LIN {X 0,Y 373.956,Z 1100.228,A -85,B 0,C 180,E1 19319.905,E2 19319.905} C_VEL
LIN {X 0,Y 365.783,Z 1123.311,A -85,B 0,C 180,E1 19326.825,E2 19326.825} C_VEL
LIN {X 0,Y 361.232,Z 1139.651,A -85,B 0,C 180,E1 19333.998,E2 19333.998} C_VEL
LIN {X 0,Y 359.65,Z 1148.795,A -85,B 0,C 180,E1 19340.296,E2 19340.296} C_VEL
LIN {X 0,Y 359.245,Z 1152.82,A -85,B 0,C 180,E1 19345.159,E2 19345.159} C_VEL
LIN {X 0,Y 359.425,Z 1154.198,A -85,B 0,C 180,E1 19349.998,E2 19349.998} C_VEL
LIN {X 0,Y 359.256,Z 1152.829,A -85,B 0,C 180,E1 19354.837,E2 19354.837} C_VEL
LIN {X 0,Y 359.821,Z 1147.421,A -85,B 0,C 180,E1 19360.921,E2 19360.921} C_VEL
LIN {X 0,Y 362.025,Z 1136.467,A -85,B 0,C 180,E1 19367.662,E2 19367.662} C_VEL
LIN {X 0,Y 366.908,Z 1119.796,A -85,B 0,C 180,E1 19374.388,E2 19374.388} C_VEL
LIN {X 0,Y 374.76,Z 1097.852,A -85,B 0,C 180,E1 19380.69,E2 19380.69} C_VEL
LIN {X 0,Y 385.507,Z 1070.168,A -85,B 0,C 180,E1 19386.483,E2 19386.483} C_VEL
LIN {X 0,Y 398.345,Z 1037.029,A -85,B 0,C 180,E1 19391.528,E2 19391.528} C_VEL
LIN {X 0,Y 411.863,Z 998.645,A -85,B 0,C 180,E1 19395.754,E2 19395.754} C_VEL
LIN {X 0,Y 424.268,Z 957.523,A -85,B 0,C 180,E1 19398.972,E2 19398.972} C_VEL
LIN {X 0,Y 433.607,Z 917.598,A -85,B 0,C 180,E1 19401.2,E2 19401.2} C_VEL
LIN {X 0,Y 431.056,Z 908.486,A -85,B 0,C 180,E1 19402.307,E2 19402.307} C_VEL
LIN {X 0,Y 426.576,Z 900.935,A -85,B 0,C 180,E1 19403.608,E2 19403.608} C_VEL
LIN {X 0,Y 417.797,Z 890.205,A -85,B 0,C 180,E1 19405.959,E2 19405.959} C_VEL
LIN {X 0,Y 405.491,Z 863.569,A -85,B 0,C 180,E1 19410.288,E2 19410.288} C_VEL
LIN {X 0,Y 391.387,Z 839.153,A -85,B 0,C 180,E1 19415.267,E2 19415.267} C_VEL
LIN {X 0,Y 377.889,Z 819.617,A -85,B 0,C 180,E1 19420.846,E2 19420.846} C_VEL
LIN {X 0,Y 371.927,Z 812.012,A -85,B 0,C 180,E1 19423.898,E2 19423.898} C_VEL
LIN {X 0,Y 367.631,Z 805.669,A -85,B 0,C 180,E1 19426.606,E2 19426.606} C_VEL
LIN {X 0,Y 363.551,Z 800.282,A -85,B 0,C 180,E1 19429.732,E2 19429.732} C_VEL
LIN {X 0,Y 362.215,Z 798.402,A -85,B 0,C 180,E1 19430.985,E2 19430.985} C_VEL
LIN {X 0,Y 357.922,Z 792.601,A -85,B 0,C 180,E1 19436.9,E2 19436.9} C_VEL
LIN {X 0,Y 357.785,Z 791.099,A -85,B 0,C 180,E1 19437.582,E2 19437.582} C_VEL
LIN {X 0,Y 357.664,Z 791.872,A -85,B 0,C 180,E1 19445.486,E2 19445.486} C_VEL
LIN {X 0,Y 360.859,Z 797.744,A -85,B 0,C 180,E1 19450.899,E2 19450.899} C_VEL
LIN {X 0,Y 363.277,Z 799.765,A -85,B 0,C 180,E1 19453.203,E2 19453.203} C_VEL
LIN {X 0,Y 366.794,Z 805.247,A -85,B 0,C 180,E1 19456.044,E2 19456.044} C_VEL
LIN {X 0,Y 368.948,Z 807.739,A -85,B 0,C 180,E1 19457.467,E2 19457.467} C_VEL
LIN {X 0,Y 374.683,Z 815.764,A -85,B 0,C 180,E1 19460.76,E2 19460.76} C_VEL
LIN {X 0,Y 383.493,Z 827.748,A -85,B 0,C 180,E1 19464.796,E2 19464.796} C_VEL
LIN {X 0,Y 398.322,Z 850.048,A -85,B 0,C 180,E1 19470.272,E2 19470.272} C_VEL
LIN {X 0,Y 412.31,Z 876.094,A -85,B 0,C 180,E1 19475.03,E2 19475.03} C_VEL
LIN {X 0,Y 424.367,Z 905.945,A -85,B 0,C 180,E1 19479.392,E2 19479.392} C_VEL
LIN {X 0,Y 428.186,Z 921.116,A -85,B 0,C 180,E1 19481.238,E2 19481.238} C_VEL
LIN {X 0,Y 417.887,Z 960.689,A -85,B 0,C 180,E1 19483.521,E2 19483.521} C_VEL
LIN {X 0,Y 406.177,Z 996.477,A -85,B 0,C 180,E1 19486.442,E2 19486.442} C_VEL
LIN {X 0,Y 392.908,Z 1031.099,A -85,B 0,C 180,E1 19490.39,E2 19490.39} C_VEL
LIN {X 0,Y 380.116,Z 1061.22,A -85,B 0,C 180,E1 19495.164,E2 19495.164} C_VEL
LIN {X 0,Y 368.183,Z 1087.867,A -85,B 0,C 180,E1 19501.085,E2 19501.085} C_VEL
LIN {X 0,Y 359.507,Z 1108.593,A -85,B 0,C 180,E1 19507.711,E2 19507.711} C_VEL
LIN {X 0,Y 354.448,Z 1122.693,A -85,B 0,C 180,E1 19514.392,E2 19514.392} C_VEL
LIN {X 0,Y 352.341,Z 1130.443,A -85,B 0,C 180,E1 19520.097,E2 19520.097} C_VEL
LIN {X 0,Y 351.551,Z 1134.292,A -85,B 0,C 180,E1 19525.057,E2 19525.057} C_VEL
LIN {X 0,Y 351.584,Z 1135.551,A -85,B 0,C 180,E1 19530.002,E2 19530.002} C_VEL
LIN {X 0,Y 351.61,Z 1134.245,A -85,B 0,C 180,E1 19534.946,E2 19534.946} C_VEL
LIN {X 0,Y 352.649,Z 1128.889,A -85,B 0,C 180,E1 19541.15,E2 19541.15} C_VEL
LIN {X 0,Y 355.894,Z 1118.129,A -85,B 0,C 180,E1 19547.981,E2 19547.981} C_VEL
LIN {X 0,Y 362.33,Z 1101.558,A -85,B 0,C 180,E1 19554.721,E2 19554.721} C_VEL
LIN {X 0,Y 372.526,Z 1078.136,A -85,B 0,C 180,E1 19561.211,E2 19561.211} C_VEL
LIN {X 0,Y 384.637,Z 1050.732,A -85,B 0,C 180,E1 19566.572,E2 19566.572} C_VEL
LIN {X 0,Y 398.251,Z 1017.644,A -85,B 0,C 180,E1 19571.2,E2 19571.2} C_VEL
LIN {X 0,Y 411.718,Z 980.096,A -85,B 0,C 180,E1 19574.923,E2 19574.923} C_VEL
LIN {X 0,Y 423.676,Z 939.446,A -85,B 0,C 180,E1 19577.719,E2 19577.719} C_VEL
LIN {X 0,Y 428.181,Z 918.706,A -85,B 0,C 180,E1 19578.835,E2 19578.835} C_VEL
LIN {X 0,Y 417.88,Z 888.908,A -85,B 0,C 180,E1 19582.883,E2 19582.883} C_VEL
LIN {X 0,Y 404.192,Z 860.481,A -85,B 0,C 180,E1 19587.547,E2 19587.547} C_VEL
LIN {X 0,Y 389.923,Z 837.253,A -85,B 0,C 180,E1 19592.513,E2 19592.513} C_VEL
LIN {X 0,Y 377.483,Z 819.326,A -85,B 0,C 180,E1 19597.664,E2 19597.664} C_VEL
LIN {X 0,Y 372.107,Z 812.286,A -85,B 0,C 180,E1 19600.401,E2 19600.401} C_VEL
LIN {X 0,Y 367.521,Z 805.745,A -85,B 0,C 180,E1 19603.219,E2 19603.219} C_VEL
LIN {X 0,Y 363.319,Z 800.256,A -85,B 0,C 180,E1 19606.402,E2 19606.402} C_VEL
LIN {X 0,Y 362.197,Z 798.481,A -85,B 0,C 180,E1 19607.448,E2 19607.448} C_VEL
LIN {X 0,Y 357.808,Z 792.997,A -85,B 0,C 180,E1 19613.093,E2 19613.093} C_VEL
LIN {X 0,Y 357.566,Z 791.207,A -85,B 0,C 180,E1 19613.969,E2 19613.969} C_VEL
LIN {X 0,Y 357.77,Z 791.665,A -85,B 0,C 180,E1 19623.253,E2 19623.253} C_VEL
LIN {X 0,Y 360.689,Z 797.51,A -85,B 0,C 180,E1 19627.837,E2 19627.837} C_VEL
LIN {X 0,Y 363.41,Z 799.856,A -85,B 0,C 180,E1 19630.348,E2 19630.348} C_VEL
LIN {X 0,Y 367.37,Z 805.514,A -85,B 0,C 180,E1 19633.404,E2 19633.404} C_VEL
LIN {X 0,Y 369.332,Z 808.368,A -85,B 0,C 180,E1 19634.694,E2 19634.694} C_VEL
LIN {X 0,Y 374.696,Z 815.689,A -85,B 0,C 180,E1 19637.72,E2 19637.72} C_VEL
LIN {X 0,Y 383.778,Z 828.216,A -85,B 0,C 180,E1 19641.864,E2 19641.864} C_VEL
LIN {X 0,Y 397.292,Z 848.846,A -85,B 0,C 180,E1 19646.917,E2 19646.917} C_VEL
LIN {X 0,Y 411.35,Z 875.442,A -85,B 0,C 180,E1 19651.804,E2 19651.804} C_VEL
LIN {X 0,Y 423.261,Z 905.411,A -85,B 0,C 180,E1 19656.19,E2 19656.19} C_VEL
LIN {X 0,Y 427.768,Z 921.449,A -85,B 0,C 180,E1 19658.22,E2 19658.22} C_VEL
LIN {X 0,Y 417.52,Z 961.645,A -85,B 0,C 180,E1 19660.513,E2 19660.513} C_VEL
LIN {X 0,Y 405.27,Z 1000.897,A -85,B 0,C 180,E1 19663.695,E2 19663.695} C_VEL
LIN {X 0,Y 391.626,Z 1038.299,A -85,B 0,C 180,E1 19667.909,E2 19667.909} C_VEL
LIN {X 0,Y 378.356,Z 1071.449,A -85,B 0,C 180,E1 19673.078,E2 19673.078} C_VEL
LIN {X 0,Y 366.86,Z 1099.983,A -85,B 0,C 180,E1 19679.261,E2 19679.261} C_VEL
LIN {X 0,Y 358.287,Z 1123.082,A -85,B 0,C 180,E1 19686.31,E2 19686.31} C_VEL
LIN {X 0,Y 353.392,Z 1139.77,A -85,B 0,C 180,E1 19693.816,E2 19693.816} C_VEL
LIN {X 0,Y 351.787,Z 1148.584,A -85,B 0,C 180,E1 19700.077,E2 19700.077} C_VEL
LIN {X 0,Y 351.344,Z 1152.612,A -85,B 0,C 180,E1 19705.05,E2 19705.05} C_VEL
LIN {X 0,Y 351.526,Z 1153.991,A -85,B 0,C 180,E1 19709.998,E2 19709.998} C_VEL
LIN {X 0,Y 351.354,Z 1152.621,A -85,B 0,C 180,E1 19714.946,E2 19714.946} C_VEL
LIN {X 0,Y 351.953,Z 1147.208,A -85,B 0,C 180,E1 19721.168,E2 19721.168} C_VEL
LIN {X 0,Y 354.33,Z 1136.25,A -85,B 0,C 180,E1 19728.058,E2 19728.058} C_VEL
LIN {X 0,Y 359.478,Z 1119.569,A -85,B 0,C 180,E1 19734.926,E2 19734.926} C_VEL
LIN {X 0,Y 367.707,Z 1097.609,A -85,B 0,C 180,E1 19741.345,E2 19741.345} C_VEL
LIN {X 0,Y 378.945,Z 1069.961,A -85,B 0,C 180,E1 19747.209,E2 19747.209} C_VEL
LIN {X 0,Y 392.299,Z 1036.729,A -85,B 0,C 180,E1 19752.316,E2 19752.316} C_VEL
LIN {X 0,Y 406.23,Z 998.283,A -85,B 0,C 180,E1 19756.577,E2 19756.577} C_VEL
LIN {X 0,Y 419.021,Z 957.147,A -85,B 0,C 180,E1 19759.799,E2 19759.799} C_VEL
LIN {X 0,Y 427.819,Z 920.28,A -85,B 0,C 180,E1 19761.9,E2 19761.9} C_VEL
LIN {X 0,Y 417.931,Z 890.491,A -85,B 0,C 180,E1 19765.913,E2 19765.913} C_VEL
LIN {X 0,Y 417.797,Z 890.205,A -85,B 0,C 180,E1 19765.959,E2 19765.959} C_VEL
LIN {X 0,Y 414.753,Z 885.487,A -85,B 0,C 180,E1 19766.885,E2 19766.885} C_VEL
LIN {X 0,Y 404.818,Z 875.598,A -85,B 0,C 180,E1 19769.67,E2 19769.67} C_VEL
LIN {X 0,Y 404.141,Z 874.327,A -85,B 0,C 180,E1 19769.908,E2 19769.908} C_VEL
LIN {X 0,Y 390.792,Z 849.549,A -85,B 0,C 180,E1 19774.923,E2 19774.923} C_VEL
LIN {X 0,Y 379.056,Z 831.63,A -85,B 0,C 180,E1 19779.768,E2 19779.768} C_VEL
LIN {X 0,Y 370.576,Z 819.735,A -85,B 0,C 180,E1 19784.066,E2 19784.066} C_VEL
LIN {X 0,Y 365.782,Z 813.016,A -85,B 0,C 180,E1 19787.146,E2 19787.146} C_VEL
LIN {X 0,Y 361.886,Z 806.955,A -85,B 0,C 180,E1 19790.369,E2 19790.369} C_VEL
LIN {X 0,Y 356.82,Z 800.076,A -85,B 0,C 180,E1 19797.271,E2 19797.271} C_VEL
LIN {X 0,Y 356.387,Z 798.849,A -85,B 0,C 180,E1 19798.791,E2 19798.791} C_VEL
LIN {X 0,Y 356.618,Z 799.725,A -85,B 0,C 180,E1 19805.296,E2 19805.296} C_VEL
LIN {X 0,Y 359.918,Z 805.614,A -85,B 0,C 180,E1 19810.928,E2 19810.928} C_VEL
LIN {X 0,Y 361.974,Z 807.59,A -85,B 0,C 180,E1 19812.943,E2 19812.943} C_VEL
LIN {X 0,Y 365.87,Z 813.166,A -85,B 0,C 180,E1 19816.086,E2 19816.086} C_VEL
LIN {X 0,Y 373.131,Z 823.471,A -85,B 0,C 180,E1 19820.507,E2 19820.507} C_VEL
LIN {X 0,Y 381.532,Z 835.16,A -85,B 0,C 180,E1 19824.45,E2 19824.45} C_VEL
LIN {X 0,Y 395.223,Z 856.602,A -85,B 0,C 180,E1 19829.82,E2 19829.82} C_VEL
LIN {X 0,Y 408.571,Z 882.567,A -85,B 0,C 180,E1 19834.645,E2 19834.645} C_VEL
LIN {X 0,Y 419.409,Z 910.851,A -85,B 0,C 180,E1 19838.886,E2 19838.886} C_VEL
LIN {X 0,Y 422.643,Z 923.525,A -85,B 0,C 180,E1 19840.525,E2 19840.525} C_VEL
LIN {X 0,Y 411.782,Z 963.336,A -85,B 0,C 180,E1 19842.877,E2 19842.877} C_VEL
LIN {X 0,Y 399.286,Z 999.96,A -85,B 0,C 180,E1 19845.975,E2 19845.975} C_VEL
LIN {X 0,Y 386.152,Z 1032.812,A -85,B 0,C 180,E1 19849.836,E2 19849.836} C_VEL
LIN {X 0,Y 373.24,Z 1062.126,A -85,B 0,C 180,E1 19854.592,E2 19854.592} C_VEL
LIN {X 0,Y 361.146,Z 1088.094,A -85,B 0,C 180,E1 19860.467,E2 19860.467} C_VEL
LIN {X 0,Y 352.084,Z 1108.811,A -85,B 0,C 180,E1 19867.215,E2 19867.215} C_VEL
LIN {X 0,Y 346.742,Z 1122.898,A -85,B 0,C 180,E1 19874.031,E2 19874.031} C_VEL
LIN {X 0,Y 344.182,Z 1131.817,A -85,B 0,C 180,E1 19881.139,E2 19881.139} C_VEL
LIN {X 0,Y 343.604,Z 1135.449,A -85,B 0,C 180,E1 19887.475,E2 19887.475} C_VEL
LIN {X 0,Y 343.67,Z 1135.428,A -85,B 0,C 180,E1 19892.529,E2 19892.529} C_VEL
LIN {X 0,Y 344.122,Z 1132.272,A -85,B 0,C 180,E1 19898.251,E2 19898.251} C_VEL
LIN {X 0,Y 346.349,Z 1123.943,A -85,B 0,C 180,E1 19905.22,E2 19905.22} C_VEL
LIN {X 0,Y 352.168,Z 1108.548,A -85,B 0,C 180,E1 19912.784,E2 19912.784} C_VEL
LIN {X 0,Y 361.342,Z 1087.725,A -85,B 0,C 180,E1 19919.52,E2 19919.52} C_VEL
LIN {X 0,Y 373.954,Z 1060.341,A -85,B 0,C 180,E1 19925.646,E2 19925.646} C_VEL
LIN {X 0,Y 388.096,Z 1028.24,A -85,B 0,C 180,E1 19930.669,E2 19930.669} C_VEL
LIN {X 0,Y 402.094,Z 992.251,A -85,B 0,C 180,E1 19934.66,E2 19934.66} C_VEL
LIN {X 0,Y 414.776,Z 953.143,A -85,B 0,C 180,E1 19937.711,E2 19937.711} C_VEL
LIN {X 0,Y 422.617,Z 922.16,A -85,B 0,C 180,E1 19939.467,E2 19939.467} C_VEL
LIN {X 0,Y 412.652,Z 892.425,A -85,B 0,C 180,E1 19943.666,E2 19943.666} C_VEL
LIN {X 0,Y 400.208,Z 865.768,A -85,B 0,C 180,E1 19948.226,E2 19948.226} C_VEL
LIN {X 0,Y 386.717,Z 843.189,A -85,B 0,C 180,E1 19953.213,E2 19953.213} C_VEL
LIN {X 0,Y 375.38,Z 826.412,A -85,B 0,C 180,E1 19958.148,E2 19958.148} C_VEL
LIN {X 0,Y 370.2,Z 819.464,A -85,B 0,C 180,E1 19960.88,E2 19960.88} C_VEL
LIN {X 0,Y 365.691,Z 813.099,A -85,B 0,C 180,E1 19963.752,E2 19963.752} C_VEL
LIN {X 0,Y 361.772,Z 807.296,A -85,B 0,C 180,E1 19966.913,E2 19966.913} C_VEL
LIN {X 0,Y 356.662,Z 800.295,A -85,B 0,C 180,E1 19973.552,E2 19973.552} C_VEL
LIN {X 0,Y 356.158,Z 798.839,A -85,B 0,C 180,E1 19975.11,E2 19975.11} C_VEL
LIN {X 0,Y 356.714,Z 799.636,A -85,B 0,C 180,E1 19983.11,E2 19983.11} C_VEL
LIN {X 0,Y 360.019,Z 805.576,A -85,B 0,C 180,E1 19988.156,E2 19988.156} C_VEL
LIN {X 0,Y 362.076,Z 807.594,A -85,B 0,C 180,E1 19990.082,E2 19990.082} C_VEL
LIN {X 0,Y 366.184,Z 813.294,A -85,B 0,C 180,E1 19993.296,E2 19993.296} C_VEL
LIN {X 0,Y 373.149,Z 823.441,A -85,B 0,C 180,E1 19997.491,E2 19997.491} C_VEL
LIN {X 0,Y 381.743,Z 835.576,A -85,B 0,C 180,E1 20001.528,E2 20001.528} C_VEL
LIN {X 0,Y 394.839,Z 856.498,A -85,B 0,C 180,E1 20006.712,E2 20006.712} C_VEL
LIN {X 0,Y 408.266,Z 883.5,A -85,B 0,C 180,E1 20011.681,E2 20011.681} C_VEL
LIN {X 0,Y 418.825,Z 911.999,A -85,B 0,C 180,E1 20015.909,E2 20015.909} C_VEL
LIN {X 0,Y 421.842,Z 925.41,A -85,B 0,C 180,E1 20017.579,E2 20017.579} C_VEL
LIN {X 0,Y 410.357,Z 967.994,A -85,B 0,C 180,E1 20020.141,E2 20020.141} C_VEL
LIN {X 0,Y 397.869,Z 1005.569,A -85,B 0,C 180,E1 20023.349,E2 20023.349} C_VEL
LIN {X 0,Y 384.76,Z 1040.072,A -85,B 0,C 180,E1 20027.384,E2 20027.384} C_VEL
LIN {X 0,Y 371.326,Z 1072.396,A -85,B 0,C 180,E1 20032.554,E2 20032.554} C_VEL
LIN {X 0,Y 359.735,Z 1099.736,A -85,B 0,C 180,E1 20038.583,E2 20038.583} C_VEL
LIN {X 0,Y 351.295,Z 1121.451,A -85,B 0,C 180,E1 20045.277,E2 20045.277} C_VEL
LIN {X 0,Y 346.242,Z 1137.175,A -85,B 0,C 180,E1 20052.16,E2 20052.16} C_VEL
LIN {X 0,Y 344.148,Z 1146.969,A -85,B 0,C 180,E1 20058.571,E2 20058.571} C_VEL
LIN {X 0,Y 343.457,Z 1152.404,A -85,B 0,C 180,E1 20064.936,E2 20064.936} C_VEL
LIN {X 0,Y 343.654,Z 1153.784,A -85,B 0,C 180,E1 20069.998,E2 20069.998} C_VEL
LIN {X 0,Y 343.464,Z 1152.414,A -85,B 0,C 180,E1 20075.059,E2 20075.059} C_VEL
LIN {X 0,Y 344.118,Z 1146.997,A -85,B 0,C 180,E1 20081.426,E2 20081.426} C_VEL
LIN {X 0,Y 346.636,Z 1136.033,A -85,B 0,C 180,E1 20088.473,E2 20088.473} C_VEL
LIN {X 0,Y 352.107,Z 1119.343,A -85,B 0,C 180,E1 20095.485,E2 20095.485} C_VEL
LIN {X 0,Y 360.712,Z 1097.368,A -85,B 0,C 180,E1 20102.024,E2 20102.024} C_VEL
LIN {X 0,Y 372.498,Z 1069.702,A -85,B 0,C 180,E1 20107.965,E2 20107.965} C_VEL
LIN {X 0,Y 386.02,Z 1037.209,A -85,B 0,C 180,E1 20113.03,E2 20113.03} C_VEL
LIN {X 0,Y 400.418,Z 998.783,A -85,B 0,C 180,E1 20117.342,E2 20117.342} C_VEL
LIN {X 0,Y 413.86,Z 956.676,A -85,B 0,C 180,E1 20120.657,E2 20120.657} C_VEL
LIN {X 0,Y 422.114,Z 923.436,A -85,B 0,C 180,E1 20122.577,E2 20122.577} C_VEL
LIN {X 0,Y 412.89,Z 894.546,A -85,B 0,C 180,E1 20126.615,E2 20126.615} C_VEL
LIN {X 0,Y 404.141,Z 874.327,A -85,B 0,C 180,E1 20129.908,E2 20129.908} C_VEL
LIN {X 0,Y 399.335,Z 868.608,A -85,B 0,C 180,E1 20131.445,E2 20131.445} C_VEL
LIN {X 0,Y 390.73,Z 861.226,A -85,B 0,C 180,E1 20134.206,E2 20134.206} C_VEL
LIN {X 0,Y 377.96,Z 840.111,A -85,B 0,C 180,E1 20139.686,E2 20139.686} C_VEL
LIN {X 0,Y 368.6,Z 826.875,A -85,B 0,C 180,E1 20144.59,E2 20144.59} C_VEL
LIN {X 0,Y 364.127,Z 820.46,A -85,B 0,C 180,E1 20147.577,E2 20147.577} C_VEL
LIN {X 0,Y 359.657,Z 813.776,A -85,B 0,C 180,E1 20151.531,E2 20151.531} C_VEL
LIN {X 0,Y 355.734,Z 807.55,A -85,B 0,C 180,E1 20157.645,E2 20157.645} C_VEL
LIN {X 0,Y 355.545,Z 807.004,A -85,B 0,C 180,E1 20164.827,E2 20164.827} C_VEL
LIN {X 0,Y 358.431,Z 813.129,A -85,B 0,C 180,E1 20170.358,E2 20170.358} C_VEL
LIN {X 0,Y 360.688,Z 815.356,A -85,B 0,C 180,E1 20172.684,E2 20172.684} C_VEL
LIN {X 0,Y 365.08,Z 821.214,A -85,B 0,C 180,E1 20176.218,E2 20176.218} C_VEL
LIN {X 0,Y 375.393,Z 836.314,A -85,B 0,C 180,E1 20182.189,E2 20182.189} C_VEL
LIN {X 0,Y 387.289,Z 855.022,A -85,B 0,C 180,E1 20187.452,E2 20187.452} C_VEL
LIN {X 0,Y 400.473,Z 879.378,A -85,B 0,C 180,E1 20192.594,E2 20192.594} C_VEL
LIN {X 0,Y 411.5,Z 906.731,A -85,B 0,C 180,E1 20197.086,E2 20197.086} C_VEL
LIN {X 0,Y 416.82,Z 926.983,A -85,B 0,C 180,E1 20199.841,E2 20199.841} C_VEL
LIN {X 0,Y 405.157,Z 967.996,A -85,B 0,C 180,E1 20202.37,E2 20202.37} C_VEL
LIN {X 0,Y 391.2,Z 1006.522,A -85,B 0,C 180,E1 20205.803,E2 20205.803} C_VEL
LIN {X 0,Y 376.331,Z 1041.514,A -85,B 0,C 180,E1 20210.274,E2 20210.274} C_VEL
LIN {X 0,Y 362.524,Z 1071.16,A -85,B 0,C 180,E1 20215.654,E2 20215.654} C_VEL
LIN {X 0,Y 351.163,Z 1094.685,A -85,B 0,C 180,E1 20221.668,E2 20221.668} C_VEL
LIN {X 0,Y 342.795,Z 1113.426,A -85,B 0,C 180,E1 20228.581,E2 20228.581} C_VEL
LIN {X 0,Y 337.973,Z 1126.183,A -85,B 0,C 180,E1 20235.728,E2 20235.728} C_VEL
LIN {X 0,Y 336.036,Z 1133.453,A -85,B 0,C 180,E1 20242.766,E2 20242.766} C_VEL
LIN {X 0,Y 335.816,Z 1135.964,A -85,B 0,C 180,E1 20250.002,E2 20250.002} C_VEL
LIN {X 0,Y 336.06,Z 1133.36,A -85,B 0,C 180,E1 20257.265,E2 20257.265} C_VEL
LIN {X 0,Y 338.002,Z 1126.018,A -85,B 0,C 180,E1 20264.276,E2 20264.276} C_VEL
LIN {X 0,Y 342.836,Z 1113.143,A -85,B 0,C 180,E1 20271.43,E2 20271.43} C_VEL
LIN {X 0,Y 351.323,Z 1094.322,A -85,B 0,C 180,E1 20278.323,E2 20278.323} C_VEL
LIN {X 0,Y 363.343,Z 1069.311,A -85,B 0,C 180,E1 20284.625,E2 20284.625} C_VEL
LIN {X 0,Y 377.374,Z 1039.079,A -85,B 0,C 180,E1 20289.974,E2 20289.974} C_VEL
LIN {X 0,Y 391.487,Z 1005.73,A -85,B 0,C 180,E1 20294.161,E2 20294.161} C_VEL
LIN {X 0,Y 405.077,Z 967.625,A -85,B 0,C 180,E1 20297.565,E2 20297.565} C_VEL
LIN {X 0,Y 416.93,Z 925.155,A -85,B 0,C 180,E1 20300.186,E2 20300.186} C_VEL
LIN {X 0,Y 408.009,Z 897.317,A -85,B 0,C 180,E1 20304.251,E2 20304.251} C_VEL
LIN {X 0,Y 396.217,Z 871.218,A -85,B 0,C 180,E1 20308.854,E2 20308.854} C_VEL
LIN {X 0,Y 382.482,Z 846.984,A -85,B 0,C 180,E1 20314.396,E2 20314.396} C_VEL
LIN {X 0,Y 369.715,Z 827.919,A -85,B 0,C 180,E1 20320.592,E2 20320.592} C_VEL
LIN {X 0,Y 363.907,Z 820.37,A -85,B 0,C 180,E1 20324.29,E2 20324.29} C_VEL
LIN {X 0,Y 359.606,Z 813.888,A -85,B 0,C 180,E1 20328.023,E2 20328.023} C_VEL
LIN {X 0,Y 355.597,Z 808.076,A -85,B 0,C 180,E1 20333.774,E2 20333.774} C_VEL
LIN {X 0,Y 355.201,Z 806.676,A -85,B 0,C 180,E1 20335.097,E2 20335.097} C_VEL
LIN {X 0,Y 355.644,Z 807.427,A -85,B 0,C 180,E1 20342.89,E2 20342.89} C_VEL
LIN {X 0,Y 359.055,Z 813.453,A -85,B 0,C 180,E1 20348.178,E2 20348.178} C_VEL
LIN {X 0,Y 360.895,Z 815.689,A -85,B 0,C 180,E1 20349.963,E2 20349.963} C_VEL
LIN {X 0,Y 366.111,Z 823.182,A -85,B 0,C 180,E1 20353.985,E2 20353.985} C_VEL
LIN {X 0,Y 372.27,Z 832.124,A -85,B 0,C 180,E1 20357.61,E2 20357.61} C_VEL
LIN {X 0,Y 382.588,Z 847.392,A -85,B 0,C 180,E1 20362.472,E2 20362.472} C_VEL
LIN {X 0,Y 394.763,Z 869.006,A -85,B 0,C 180,E1 20367.49,E2 20367.49} C_VEL
LIN {X 0,Y 406.917,Z 896.393,A -85,B 0,C 180,E1 20372.348,E2 20372.348} C_VEL
LIN {X 0,Y 415.804,Z 924.576,A -85,B 0,C 180,E1 20376.473,E2 20376.473} C_VEL
LIN {X 0,Y 416.016,Z 929.066,A -85,B 0,C 180,E1 20376.922,E2 20376.922} C_VEL
LIN {X 0,Y 404.054,Z 971.469,A -85,B 0,C 180,E1 20379.55,E2 20379.55} C_VEL
LIN {X 0,Y 389.795,Z 1012.29,A -85,B 0,C 180,E1 20383.209,E2 20383.209} C_VEL
LIN {X 0,Y 375.215,Z 1048.426,A -85,B 0,C 180,E1 20387.78,E2 20387.78} C_VEL
LIN {X 0,Y 360.938,Z 1080.916,A -85,B 0,C 180,E1 20393.516,E2 20393.516} C_VEL
LIN {X 0,Y 349.381,Z 1107.786,A -85,B 0,C 180,E1 20400.229,E2 20400.229} C_VEL
LIN {X 0,Y 341.061,Z 1128.977,A -85,B 0,C 180,E1 20407.812,E2 20407.812} C_VEL
LIN {X 0,Y 337.233,Z 1142.073,A -85,B 0,C 180,E1 20414.807,E2 20414.807} C_VEL
LIN {X 0,Y 335.925,Z 1149.422,A -85,B 0,C 180,E1 20420.915,E2 20420.915} C_VEL
LIN {X 0,Y 335.614,Z 1153.221,A -85,B 0,C 180,E1 20427.41,E2 20427.41} C_VEL
LIN {X 0,Y 335.62,Z 1153.224,A -85,B 0,C 180,E1 20432.585,E2 20432.585} C_VEL
LIN {X 0,Y 335.886,Z 1149.445,A -85,B 0,C 180,E1 20439.082,E2 20439.082} C_VEL
LIN {X 0,Y 337.653,Z 1140.439,A -85,B 0,C 180,E1 20446.285,E2 20446.285} C_VEL
LIN {X 0,Y 342.184,Z 1125.878,A -85,B 0,C 180,E1 20453.483,E2 20453.483} C_VEL
LIN {X 0,Y 350.218,Z 1105.709,A -85,B 0,C 180,E1 20460.382,E2 20460.382} C_VEL
LIN {X 0,Y 360.885,Z 1081.071,A -85,B 0,C 180,E1 20466.478,E2 20466.478} C_VEL
LIN {X 0,Y 375.169,Z 1048.682,A -85,B 0,C 180,E1 20472.205,E2 20472.205} C_VEL
LIN {X 0,Y 389.849,Z 1012.531,A -85,B 0,C 180,E1 20476.777,E2 20476.777} C_VEL
LIN {X 0,Y 403.924,Z 972.317,A -85,B 0,C 180,E1 20480.395,E2 20480.395} C_VEL
LIN {X 0,Y 415.635,Z 931.022,A -85,B 0,C 180,E1 20482.989,E2 20482.989} C_VEL
LIN {X 0,Y 416.25,Z 925.64,A -85,B 0,C 180,E1 20483.394,E2 20483.394} C_VEL
LIN {X 0,Y 407.686,Z 897.989,A -85,B 0,C 180,E1 20487.405,E2 20487.405} C_VEL
LIN {X 0,Y 395.73,Z 870.912,A -85,B 0,C 180,E1 20492.187,E2 20492.187} C_VEL
LIN {X 0,Y 390.73,Z 861.226,A -85,B 0,C 180,E1 20494.206,E2 20494.206} C_VEL
LIN {X 0,Y 384.238,Z 856.089,A -85,B 0,C 180,E1 20496.492,E2 20496.492} C_VEL
LIN {X 0,Y 378.199,Z 851.399,A -85,B 0,C 180,E1 20498.883,E2 20498.883} C_VEL
LIN {X 0,Y 367.965,Z 835.3,A -85,B 0,C 180,E1 20504.333,E2 20504.333} C_VEL
LIN {X 0,Y 362.594,Z 827.934,A -85,B 0,C 180,E1 20507.95,E2 20507.95} C_VEL
LIN {X 0,Y 358.403,Z 821.505,A -85,B 0,C 180,E1 20511.79,E2 20511.79} C_VEL
LIN {X 0,Y 354.663,Z 815.023,A -85,B 0,C 180,E1 20518.02,E2 20518.02} C_VEL
LIN {X 0,Y 354.556,Z 815.299,A -85,B 0,C 180,E1 20524.912,E2 20524.912} C_VEL
LIN {X 0,Y 358.034,Z 821.369,A -85,B 0,C 180,E1 20530.986,E2 20530.986} C_VEL
LIN {X 0,Y 359.573,Z 823.552,A -85,B 0,C 180,E1 20532.601,E2 20532.601} C_VEL
LIN {X 0,Y 364.697,Z 831.046,A -85,B 0,C 180,E1 20536.721,E2 20536.721} C_VEL
LIN {X 0,Y 372.984,Z 842.849,A -85,B 0,C 180,E1 20541.608,E2 20541.608} C_VEL
LIN {X 0,Y 385.449,Z 863.469,A -85,B 0,C 180,E1 20547.436,E2 20547.436} C_VEL
LIN {X 0,Y 397.664,Z 887.863,A -85,B 0,C 180,E1 20552.577,E2 20552.577} C_VEL
LIN {X 0,Y 408.103,Z 916.432,A -85,B 0,C 180,E1 20557.274,E2 20557.274} C_VEL
LIN {X 0,Y 411.32,Z 929.318,A -85,B 0,C 180,E1 20559.096,E2 20559.096} C_VEL
LIN {X 0,Y 399.832,Z 968.464,A -85,B 0,C 180,E1 20561.541,E2 20561.541} C_VEL
LIN {X 0,Y 386.033,Z 1005.643,A -85,B 0,C 180,E1 20564.854,E2 20564.854} C_VEL
LIN {X 0,Y 371.025,Z 1039.99,A -85,B 0,C 180,E1 20569.205,E2 20569.205} C_VEL
LIN {X 0,Y 356.624,Z 1070.044,A -85,B 0,C 180,E1 20574.631,E2 20574.631} C_VEL
LIN {X 0,Y 344.12,Z 1094.913,A -85,B 0,C 180,E1 20581.034,E2 20581.034} C_VEL
LIN {X 0,Y 335.309,Z 1113.645,A -85,B 0,C 180,E1 20588.078,E2 20588.078} C_VEL
LIN {X 0,Y 330.227,Z 1126.418,A -85,B 0,C 180,E1 20595.402,E2 20595.402} C_VEL
LIN {X 0,Y 328.282,Z 1133.319,A -85,B 0,C 180,E1 20602.043,E2 20602.043} C_VEL
LIN {X 0,Y 327.946,Z 1136.171,A -85,B 0,C 180,E1 20610.002,E2 20610.002} C_VEL
LIN {X 0,Y 327.963,Z 1134.868,A -85,B 0,C 180,E1 20615.304,E2 20615.304} C_VEL
LIN {X 0,Y 329.211,Z 1129.524,A -85,B 0,C 180,E1 20621.955,E2 20621.955} C_VEL
LIN {X 0,Y 333.093,Z 1118.783,A -85,B 0,C 180,E1 20629.258,E2 20629.258} C_VEL
LIN {X 0,Y 340.524,Z 1102.24,A -85,B 0,C 180,E1 20636.423,E2 20636.423} C_VEL
LIN {X 0,Y 352.19,Z 1078.73,A -85,B 0,C 180,E1 20643.276,E2 20643.276} C_VEL
LIN {X 0,Y 365.604,Z 1051.51,A -85,B 0,C 180,E1 20648.819,E2 20648.819} C_VEL
LIN {X 0,Y 380.566,Z 1018.529,A -85,B 0,C 180,E1 20653.575,E2 20653.575} C_VEL
LIN {X 0,Y 395.523,Z 980.232,A -85,B 0,C 180,E1 20657.445,E2 20657.445} C_VEL
LIN {X 0,Y 408.596,Z 939.168,A -85,B 0,C 180,E1 20660.273,E2 20660.273} C_VEL
LIN {X 0,Y 411.13,Z 927.699,A -85,B 0,C 180,E1 20660.971,E2 20660.971} C_VEL
LIN {X 0,Y 402.183,Z 899.352,A -85,B 0,C 180,E1 20665.315,E2 20665.315} C_VEL
LIN {X 0,Y 390.994,Z 874.093,A -85,B 0,C 180,E1 20670.021,E2 20670.021} C_VEL
LIN {X 0,Y 378.994,Z 852.611,A -85,B 0,C 180,E1 20675.252,E2 20675.252} C_VEL
LIN {X 0,Y 367.963,Z 835.282,A -85,B 0,C 180,E1 20680.984,E2 20680.984} C_VEL
LIN {X 0,Y 362.15,Z 827.64,A -85,B 0,C 180,E1 20684.834,E2 20684.834} C_VEL
LIN {X 0,Y 358.273,Z 821.553,A -85,B 0,C 180,E1 20688.365,E2 20688.365} C_VEL
LIN {X 0,Y 354.501,Z 815.507,A -85,B 0,C 180,E1 20694.169,E2 20694.169} C_VEL
LIN {X 0,Y 353.843,Z 814.291,A -85,B 0,C 180,E1 20699.991,E2 20699.991} C_VEL
LIN {X 0,Y 354.645,Z 815.578,A -85,B 0,C 180,E1 20702.899,E2 20702.899} C_VEL
LIN {X 0,Y 358.399,Z 821.506,A -85,B 0,C 180,E1 20708.499,E2 20708.499} C_VEL
LIN {X 0,Y 364.671,Z 830.908,A -85,B 0,C 180,E1 20713.735,E2 20713.735} C_VEL
LIN {X 0,Y 372.865,Z 842.858,A -85,B 0,C 180,E1 20718.576,E2 20718.576} C_VEL
LIN {X 0,Y 385.253,Z 863.463,A -85,B 0,C 180,E1 20724.403,E2 20724.403} C_VEL
LIN {X 0,Y 397.327,Z 888.876,A -85,B 0,C 180,E1 20729.629,E2 20729.629} C_VEL
LIN {X 0,Y 406.838,Z 915.155,A -85,B 0,C 180,E1 20733.948,E2 20733.948} C_VEL
LIN {X 0,Y 410.732,Z 930.495,A -85,B 0,C 180,E1 20736.131,E2 20736.131} C_VEL
LIN {X 0,Y 398.626,Z 972.096,A -85,B 0,C 180,E1 20738.736,E2 20738.736} C_VEL
LIN {X 0,Y 384.219,Z 1012.164,A -85,B 0,C 180,E1 20742.35,E2 20742.35} C_VEL
LIN {X 0,Y 369.1,Z 1048.381,A -85,B 0,C 180,E1 20746.962,E2 20746.962} C_VEL
LIN {X 0,Y 354.285,Z 1080.904,A -85,B 0,C 180,E1 20752.78,E2 20752.78} C_VEL
LIN {X 0,Y 342.077,Z 1108.064,A -85,B 0,C 180,E1 20759.702,E2 20759.702} C_VEL
LIN {X 0,Y 333.56,Z 1128.752,A -85,B 0,C 180,E1 20767.285,E2 20767.285} C_VEL
LIN {X 0,Y 329.261,Z 1142.746,A -85,B 0,C 180,E1 20775.038,E2 20775.038} C_VEL
LIN {X 0,Y 327.939,Z 1150.306,A -85,B 0,C 180,E1 20782.03,E2 20782.03} C_VEL
LIN {X 0,Y 327.705,Z 1153.013,A -85,B 0,C 180,E1 20787.348,E2 20787.348} C_VEL
LIN {X 0,Y 327.71,Z 1153.017,A -85,B 0,C 180,E1 20792.648,E2 20792.648} C_VEL
LIN {X 0,Y 328.018,Z 1149.235,A -85,B 0,C 180,E1 20799.301,E2 20799.301} C_VEL
LIN {X 0,Y 329.934,Z 1140.225,A -85,B 0,C 180,E1 20806.677,E2 20806.677} C_VEL
LIN {X 0,Y 334.729,Z 1125.656,A -85,B 0,C 180,E1 20814.038,E2 20814.038} C_VEL
LIN {X 0,Y 342.994,Z 1105.971,A -85,B 0,C 180,E1 20820.928,E2 20820.928} C_VEL
LIN {X 0,Y 354.229,Z 1081.056,A -85,B 0,C 180,E1 20827.216,E2 20827.216} C_VEL
LIN {X 0,Y 368.857,Z 1049.128,A -85,B 0,C 180,E1 20832.948,E2 20832.948} C_VEL
LIN {X 0,Y 384.321,Z 1012.219,A -85,B 0,C 180,E1 20837.661,E2 20837.661} C_VEL
LIN {X 0,Y 398.817,Z 971.944,A -85,B 0,C 180,E1 20841.291,E2 20841.291} C_VEL
LIN {X 0,Y 410.748,Z 929.355,A -85,B 0,C 180,E1 20844.021,E2 20844.021} C_VEL
LIN {X 0,Y 403.027,Z 903.188,A -85,B 0,C 180,E1 20847.938,E2 20847.938} C_VEL
LIN {X 0,Y 391.942,Z 876.701,A -85,B 0,C 180,E1 20852.76,E2 20852.76} C_VEL
LIN {X 0,Y 381.532,Z 857.038,A -85,B 0,C 180,E1 20857.308,E2 20857.308} C_VEL
LIN {X 0,Y 378.199,Z 851.399,A -85,B 0,C 180,E1 20858.883,E2 20858.883} C_VEL
LIN {X 0,Y 374.25,Z 849.552,A -85,B 0,C 180,E1 20860.536,E2 20860.536} C_VEL
LIN {X 0,Y 370.205,Z 848.927,A -85,B 0,C 180,E1 20862.279,E2 20862.279} C_VEL
LIN {X 0,Y 361.202,Z 835.532,A -85,B 0,C 180,E1 20868.198,E2 20868.198} C_VEL
LIN {X 0,Y 357.111,Z 829.148,A -85,B 0,C 180,E1 20872.102,E2 20872.102} C_VEL
LIN {X 0,Y 353.5,Z 822.368,A -85,B 0,C 180,E1 20878.781,E2 20878.781} C_VEL
LIN {X 0,Y 353.551,Z 823.306,A -85,B 0,C 180,E1 20884.854,E2 20884.854} C_VEL
LIN {X 0,Y 357.386,Z 829.385,A -85,B 0,C 180,E1 20891.316,E2 20891.316} C_VEL
LIN {X 0,Y 363.24,Z 838.753,A -85,B 0,C 180,E1 20896.493,E2 20896.493} C_VEL
LIN {X 0,Y 371.142,Z 850.443,A -85,B 0,C 180,E1 20901.328,E2 20901.328} C_VEL
LIN {X 0,Y 382.921,Z 870.999,A -85,B 0,C 180,E1 20907.233,E2 20907.233} C_VEL
LIN {X 0,Y 393.952,Z 894.455,A -85,B 0,C 180,E1 20912.21,E2 20912.21} C_VEL
LIN {X 0,Y 403.46,Z 922.605,A -85,B 0,C 180,E1 20916.938,E2 20916.938} C_VEL
LIN {X 0,Y 405.469,Z 933.166,A -85,B 0,C 180,E1 20918.409,E2 20918.409} C_VEL
LIN {X 0,Y 393.771,Z 971.162,A -85,B 0,C 180,E1 20920.86,E2 20920.86} C_VEL
LIN {X 0,Y 379.964,Z 1007.113,A -85,B 0,C 180,E1 20924.132,E2 20924.132} C_VEL
LIN {X 0,Y 364.428,Z 1041.443,A -85,B 0,C 180,E1 20928.566,E2 20928.566} C_VEL
LIN {X 0,Y 349.386,Z 1071.63,A -85,B 0,C 180,E1 20934.168,E2 20934.168} C_VEL
LIN {X 0,Y 336.544,Z 1096.175,A -85,B 0,C 180,E1 20940.705,E2 20940.705} C_VEL
LIN {X 0,Y 327.213,Z 1115.331,A -85,B 0,C 180,E1 20948.26,E2 20948.26} C_VEL
LIN {X 0,Y 322.425,Z 1126.81,A -85,B 0,C 180,E1 20955.175,E2 20955.175} C_VEL
LIN {X 0,Y 320.436,Z 1133.527,A -85,B 0,C 180,E1 20961.847,E2 20961.847} C_VEL
LIN {X 0,Y 320.046,Z 1136.378,A -85,B 0,C 180,E1 20970.002,E2 20970.002} C_VEL
LIN {X 0,Y 320.137,Z 1134.589,A -85,B 0,C 180,E1 20976.287,E2 20976.287} C_VEL
LIN {X 0,Y 321.898,Z 1128.228,A -85,B 0,C 180,E1 20983.615,E2 20983.615} C_VEL
LIN {X 0,Y 326.647,Z 1116.404,A -85,B 0,C 180,E1 20991.071,E2 20991.071} C_VEL
LIN {X 0,Y 334.314,Z 1100.507,A -85,B 0,C 180,E1 20997.707,E2 20997.707} C_VEL
LIN {X 0,Y 345.788,Z 1078.313,A -85,B 0,C 180,E1 21004.167,E2 21004.167} C_VEL
LIN {X 0,Y 360.202,Z 1050.085,A -85,B 0,C 180,E1 21009.905,E2 21009.905} C_VEL
LIN {X 0,Y 375.465,Z 1017.383,A -85,B 0,C 180,E1 21014.586,E2 21014.586} C_VEL
LIN {X 0,Y 390.494,Z 979.735,A -85,B 0,C 180,E1 21018.374,E2 21018.374} C_VEL
LIN {X 0,Y 403.862,Z 938.689,A -85,B 0,C 180,E1 21021.186,E2 21021.186} C_VEL
LIN {X 0,Y 405.489,Z 930.847,A -85,B 0,C 180,E1 21021.695,E2 21021.695} C_VEL
LIN {X 0,Y 397.108,Z 903.089,A -85,B 0,C 180,E1 21026.115,E2 21026.115} C_VEL
LIN {X 0,Y 386.881,Z 879.141,A -85,B 0,C 180,E1 21030.784,E2 21030.784} C_VEL
LIN {X 0,Y 376.043,Z 859.015,A -85,B 0,C 180,E1 21035.837,E2 21035.837} C_VEL
LIN {X 0,Y 366.145,Z 842.685,A -85,B 0,C 180,E1 21041.336,E2 21041.336} C_VEL
LIN {X 0,Y 360.641,Z 835.087,A -85,B 0,C 180,E1 21045.209,E2 21045.209} C_VEL
LIN {X 0,Y 356.844,Z 829.136,A -85,B 0,C 180,E1 21048.822,E2 21048.822} C_VEL
LIN {X 0,Y 353.411,Z 822.797,A -85,B 0,C 180,E1 21054.632,E2 21054.632} C_VEL
LIN {X 0,Y 353.531,Z 822.923,A -85,B 0,C 180,E1 21062.447,E2 21062.447} C_VEL
LIN {X 0,Y 357.126,Z 829.202,A -85,B 0,C 180,E1 21068.222,E2 21068.222} C_VEL
LIN {X 0,Y 363.133,Z 838.568,A -85,B 0,C 180,E1 21073.487,E2 21073.487} C_VEL
LIN {X 0,Y 371.049,Z 850.635,A -85,B 0,C 180,E1 21078.361,E2 21078.361} C_VEL
LIN {X 0,Y 382.401,Z 870.636,A -85,B 0,C 180,E1 21084.096,E2 21084.096} C_VEL
LIN {X 0,Y 393.667,Z 895.616,A -85,B 0,C 180,E1 21089.297,E2 21089.297} C_VEL
LIN {X 0,Y 402.839,Z 923.553,A -85,B 0,C 180,E1 21093.954,E2 21093.954} C_VEL
LIN {X 0,Y 405.049,Z 932.872,A -85,B 0,C 180,E1 21095.328,E2 21095.328} C_VEL
LIN {X 0,Y 392.732,Z 974.249,A -85,B 0,C 180,E1 21098.018,E2 21098.018} C_VEL
LIN {X 0,Y 378.22,Z 1013.224,A -85,B 0,C 180,E1 21101.596,E2 21101.596} C_VEL
LIN {X 0,Y 363.183,Z 1048.091,A -85,B 0,C 180,E1 21106.083,E2 21106.083} C_VEL
LIN {X 0,Y 348.13,Z 1079.928,A -85,B 0,C 180,E1 21111.814,E2 21111.814} C_VEL
LIN {X 0,Y 335.875,Z 1106.057,A -85,B 0,C 180,E1 21118.476,E2 21118.476} C_VEL
LIN {X 0,Y 327.293,Z 1125.367,A -85,B 0,C 180,E1 21125.375,E2 21125.375} C_VEL
LIN {X 0,Y 322.191,Z 1139.971,A -85,B 0,C 180,E1 21132.905,E2 21132.905} C_VEL
LIN {X 0,Y 320.18,Z 1149,A -85,B 0,C 180,E1 21140.464,E2 21140.464} C_VEL
LIN {X 0,Y 319.796,Z 1152.805,A -85,B 0,C 180,E1 21147.282,E2 21147.282} C_VEL
LIN {X 0,Y 319.801,Z 1152.809,A -85,B 0,C 180,E1 21152.713,E2 21152.713} C_VEL
LIN {X 0,Y 320.13,Z 1149.024,A -85,B 0,C 180,E1 21159.533,E2 21159.533} C_VEL
LIN {X 0,Y 322.222,Z 1140.012,A -85,B 0,C 180,E1 21167.088,E2 21167.088} C_VEL
LIN {X 0,Y 327.752,Z 1124.388,A -85,B 0,C 180,E1 21175.067,E2 21175.067} C_VEL
LIN {X 0,Y 336.609,Z 1104.344,A -85,B 0,C 180,E1 21182.057,E2 21182.057} C_VEL
LIN {X 0,Y 348.751,Z 1078.653,A -85,B 0,C 180,E1 21188.477,E2 21188.477} C_VEL
LIN {X 0,Y 363.173,Z 1048.281,A -85,B 0,C 180,E1 21193.913,E2 21193.913} C_VEL
LIN {X 0,Y 379.197,Z 1011.122,A -85,B 0,C 180,E1 21198.651,E2 21198.651} C_VEL
LIN {X 0,Y 393.759,Z 971.79,A -85,B 0,C 180,E1 21202.187,E2 21202.187} C_VEL
LIN {X 0,Y 405.256,Z 932.943,A -85,B 0,C 180,E1 21204.668,E2 21204.668} C_VEL
LIN {X 0,Y 397.847,Z 906.763,A -85,B 0,C 180,E1 21208.755,E2 21208.755} C_VEL
LIN {X 0,Y 387.311,Z 880.428,A -85,B 0,C 180,E1 21213.745,E2 21213.745} C_VEL
LIN {X 0,Y 376.216,Z 859.295,A -85,B 0,C 180,E1 21219,E2 21219} C_VEL
LIN {X 0,Y 370.205,Z 848.927,A -85,B 0,C 180,E1 21222.279,E2 21222.279} C_VEL
LIN {X 0,Y 363.113,Z 848.688,A -85,B 0,C 180,E1 21225.813,E2 21225.813} C_VEL
LIN {X 0,Y 359.42,Z 842.873,A -85,B 0,C 180,E1 21228.657,E2 21228.657} C_VEL
LIN {X 0,Y 355.802,Z 836.825,A -85,B 0,C 180,E1 21232.372,E2 21232.372} C_VEL
LIN {X 0,Y 352.537,Z 830.216,A -85,B 0,C 180,E1 21238.778,E2 21238.778} C_VEL
LIN {X 0,Y 352.53,Z 831.047,A -85,B 0,C 180,E1 21244.654,E2 21244.654} C_VEL
LIN {X 0,Y 356.847,Z 838.611,A -85,B 0,C 180,E1 21251.954,E2 21251.954} C_VEL
LIN {X 0,Y 361.979,Z 846.913,A -85,B 0,C 180,E1 21256.469,E2 21256.469} C_VEL
LIN {X 0,Y 369.002,Z 857.999,A -85,B 0,C 180,E1 21261.064,E2 21261.064} C_VEL
LIN {X 0,Y 379.947,Z 877.921,A -85,B 0,C 180,E1 21266.872,E2 21266.872} C_VEL
LIN {X 0,Y 390.288,Z 901.767,A -85,B 0,C 180,E1 21271.986,E2 21271.986} C_VEL
LIN {X 0,Y 398.505,Z 927.761,A -85,B 0,C 180,E1 21276.458,E2 21276.458} C_VEL
LIN {X 0,Y 400.066,Z 935.647,A -85,B 0,C 180,E1 21277.632,E2 21277.632} C_VEL
LIN {X 0,Y 388.065,Z 973.074,A -85,B 0,C 180,E1 21280.098,E2 21280.098} C_VEL
LIN {X 0,Y 374.478,Z 1007.406,A -85,B 0,C 180,E1 21283.26,E2 21283.26} C_VEL
LIN {X 0,Y 358.46,Z 1041.7,A -85,B 0,C 180,E1 21287.718,E2 21287.718} C_VEL
LIN {X 0,Y 342.904,Z 1071.865,A -85,B 0,C 180,E1 21293.382,E2 21293.382} C_VEL
LIN {X 0,Y 330.096,Z 1095.369,A -85,B 0,C 180,E1 21299.678,E2 21299.678} C_VEL
LIN {X 0,Y 320.422,Z 1114.13,A -85,B 0,C 180,E1 21307.027,E2 21307.027} C_VEL
LIN {X 0,Y 314.567,Z 1127.425,A -85,B 0,C 180,E1 21315.106,E2 21315.106} C_VEL
LIN {X 0,Y 312.565,Z 1133.735,A -85,B 0,C 180,E1 21321.641,E2 21321.641} C_VEL
LIN {X 0,Y 312.148,Z 1136.585,A -85,B 0,C 180,E1 21330.002,E2 21330.002} C_VEL
LIN {X 0,Y 312.191,Z 1135.284,A -85,B 0,C 180,E1 21335.573,E2 21335.573} C_VEL
LIN {X 0,Y 313.602,Z 1129.948,A -85,B 0,C 180,E1 21342.56,E2 21342.56} C_VEL
LIN {X 0,Y 317.99,Z 1119.219,A -85,B 0,C 180,E1 21350.212,E2 21350.212} C_VEL
LIN {X 0,Y 326.203,Z 1102.69,A -85,B 0,C 180,E1 21357.679,E2 21357.679} C_VEL
LIN {X 0,Y 338.439,Z 1079.953,A -85,B 0,C 180,E1 21364.589,E2 21364.589} C_VEL
LIN {X 0,Y 353.223,Z 1052.054,A -85,B 0,C 180,E1 21370.445,E2 21370.445} C_VEL
LIN {X 0,Y 369.246,Z 1019.007,A -85,B 0,C 180,E1 21375.29,E2 21375.29} C_VEL
LIN {X 0,Y 384.847,Z 981.256,A -85,B 0,C 180,E1 21379.16,E2 21379.16} C_VEL
LIN {X 0,Y 398.808,Z 939.788,A -85,B 0,C 180,E1 21382.034,E2 21382.034} C_VEL
LIN {X 0,Y 400.038,Z 934.592,A -85,B 0,C 180,E1 21382.351,E2 21382.351} C_VEL
LIN {X 0,Y 392.12,Z 907.016,A -85,B 0,C 180,E1 21386.915,E2 21386.915} C_VEL
LIN {X 0,Y 382.133,Z 882.644,A -85,B 0,C 180,E1 21391.868,E2 21391.868} C_VEL
LIN {X 0,Y 371.18,Z 861.722,A -85,B 0,C 180,E1 21397.492,E2 21397.492} C_VEL
LIN {X 0,Y 363.007,Z 848.55,A -85,B 0,C 180,E1 21402.535,E2 21402.535} C_VEL
LIN {X 0,Y 359.058,Z 842.612,A -85,B 0,C 180,E1 21405.53,E2 21405.53} C_VEL
LIN {X 0,Y 355.697,Z 836.917,A -85,B 0,C 180,E1 21408.941,E2 21408.941} C_VEL
LIN {X 0,Y 352.367,Z 830.462,A -85,B 0,C 180,E1 21414.911,E2 21414.911} C_VEL
LIN {X 0,Y 352.52,Z 830.901,A -85,B 0,C 180,E1 21422.377,E2 21422.377} C_VEL
LIN {X 0,Y 356.083,Z 837.062,A -85,B 0,C 180,E1 21428.247,E2 21428.247} C_VEL
LIN {X 0,Y 361.742,Z 846.563,A -85,B 0,C 180,E1 21433.385,E2 21433.385} C_VEL
LIN {X 0,Y 368.868,Z 858.12,A -85,B 0,C 180,E1 21438.087,E2 21438.087} C_VEL
LIN {X 0,Y 379.46,Z 877.659,A -85,B 0,C 180,E1 21443.761,E2 21443.761} C_VEL
LIN {X 0,Y 389.383,Z 901.212,A -85,B 0,C 180,E1 21448.773,E2 21448.773} C_VEL
LIN {X 0,Y 397.463,Z 926.885,A -85,B 0,C 180,E1 21453.185,E2 21453.185} C_VEL
LIN {X 0,Y 399.505,Z 936.605,A -85,B 0,C 180,E1 21454.659,E2 21454.659} C_VEL
LIN {X 0,Y 387.04,Z 976.025,A -85,B 0,C 180,E1 21457.25,E2 21457.25} C_VEL
LIN {X 0,Y 372.216,Z 1014.453,A -85,B 0,C 180,E1 21460.838,E2 21460.838} C_VEL
LIN {X 0,Y 356.472,Z 1049.672,A -85,B 0,C 180,E1 21465.464,E2 21465.464} C_VEL
LIN {X 0,Y 341.161,Z 1080.874,A -85,B 0,C 180,E1 21471.221,E2 21471.221} C_VEL
LIN {X 0,Y 328.038,Z 1107.727,A -85,B 0,C 180,E1 21478.306,E2 21478.306} C_VEL
LIN {X 0,Y 318.608,Z 1128.303,A -85,B 0,C 180,E1 21486.155,E2 21486.155} C_VEL
LIN {X 0,Y 313.7,Z 1142.313,A -85,B 0,C 180,E1 21494.276,E2 21494.276} C_VEL
LIN {X 0,Y 312.178,Z 1149.887,A -85,B 0,C 180,E1 21501.625,E2 21501.625} C_VEL
LIN {X 0,Y 311.912,Z 1152.599,A -85,B 0,C 180,E1 21507.213,E2 21507.213} C_VEL
LIN {X 0,Y 311.917,Z 1152.602,A -85,B 0,C 180,E1 21512.782,E2 21512.782} C_VEL
LIN {X 0,Y 312.255,Z 1148.814,A -85,B 0,C 180,E1 21519.776,E2 21519.776} C_VEL
LIN {X 0,Y 314.499,Z 1139.798,A -85,B 0,C 180,E1 21527.522,E2 21527.522} C_VEL
LIN {X 0,Y 320.456,Z 1123.971,A -85,B 0,C 180,E1 21535.771,E2 21535.771} C_VEL
LIN {X 0,Y 329.981,Z 1103.371,A -85,B 0,C 180,E1 21543.04,E2 21543.04} C_VEL
LIN {X 0,Y 342.274,Z 1078.669,A -85,B 0,C 180,E1 21549.271,E2 21549.271} C_VEL
LIN {X 0,Y 357.34,Z 1048.003,A -85,B 0,C 180,E1 21554.82,E2 21554.82} C_VEL
LIN {X 0,Y 373.166,Z 1012.551,A -85,B 0,C 180,E1 21559.398,E2 21559.398} C_VEL
LIN {X 0,Y 388.773,Z 971.682,A -85,B 0,C 180,E1 21563.105,E2 21563.105} C_VEL
LIN {X 0,Y 399.578,Z 935.291,A -85,B 0,C 180,E1 21565.513,E2 21565.513} C_VEL
LIN {X 0,Y 391.692,Z 907.169,A -85,B 0,C 180,E1 21570.142,E2 21570.142} C_VEL
LIN {X 0,Y 381.253,Z 881.288,A -85,B 0,C 180,E1 21575.445,E2 21575.445} C_VEL
LIN {X 0,Y 370.444,Z 860.636,A -85,B 0,C 180,E1 21581.144,E2 21581.144} C_VEL
LIN {X 0,Y 363.113,Z 848.688,A -85,B 0,C 180,E1 21585.813,E2 21585.813} C_VEL
LIN {X 0,Y 360.05,Z 848.987,A -85,B 0,C 180,E1 21587.616,E2 21587.616} C_VEL
LIN {X 0,Y 357.246,Z 849.729,A -85,B 0,C 180,E1 21589.463,E2 21589.463} C_VEL
LIN {X 0,Y 354.396,Z 844.507,A -85,B 0,C 180,E1 21592.641,E2 21592.641} C_VEL
LIN {X 0,Y 351.473,Z 838.089,A -85,B 0,C 180,E1 21598.774,E2 21598.774} C_VEL
LIN {X 0,Y 351.423,Z 838.847,A -85,B 0,C 180,E1 21604.525,E2 21604.525} C_VEL
LIN {X 0,Y 355.492,Z 846.445,A -85,B 0,C 180,E1 21611.776,E2 21611.776} C_VEL
LIN {X 0,Y 360.36,Z 854.727,A -85,B 0,C 180,E1 21616.339,E2 21616.339} C_VEL
LIN {X 0,Y 367.429,Z 866.582,A -85,B 0,C 180,E1 21621.158,E2 21621.158} C_VEL
LIN {X 0,Y 376.988,Z 885.343,A -85,B 0,C 180,E1 21626.623,E2 21626.623} C_VEL
LIN {X 0,Y 386.368,Z 908.335,A -85,B 0,C 180,E1 21631.642,E2 21631.642} C_VEL
LIN {X 0,Y 393.834,Z 934.442,A -85,B 0,C 180,E1 21636.234,E2 21636.234} C_VEL
LIN {X 0,Y 394.47,Z 939.096,A -85,B 0,C 180,E1 21636.886,E2 21636.886} C_VEL
LIN {X 0,Y 380.583,Z 980.047,A -85,B 0,C 180,E1 21639.72,E2 21639.72} C_VEL
LIN {X 0,Y 365.404,Z 1015.704,A -85,B 0,C 180,E1 21643.271,E2 21643.271} C_VEL
LIN {X 0,Y 349.476,Z 1047.928,A -85,B 0,C 180,E1 21647.83,E2 21647.83} C_VEL
LIN {X 0,Y 334.97,Z 1074.705,A -85,B 0,C 180,E1 21653.181,E2 21653.181} C_VEL
LIN {X 0,Y 322.043,Z 1097.527,A -85,B 0,C 180,E1 21659.62,E2 21659.62} C_VEL
LIN {X 0,Y 312.267,Z 1115.862,A -85,B 0,C 180,E1 21667.22,E2 21667.22} C_VEL
LIN {X 0,Y 306.854,Z 1127.636,A -85,B 0,C 180,E1 21674.723,E2 21674.723} C_VEL
LIN {X 0,Y 304.718,Z 1133.943,A -85,B 0,C 180,E1 21681.424,E2 21681.424} C_VEL
LIN {X 0,Y 304.248,Z 1136.792,A -85,B 0,C 180,E1 21690.002,E2 21690.002} C_VEL
LIN {X 0,Y 304.308,Z 1135.492,A -85,B 0,C 180,E1 21695.718,E2 21695.718} C_VEL
LIN {X 0,Y 305.824,Z 1130.159,A -85,B 0,C 180,E1 21702.885,E2 21702.885} C_VEL
LIN {X 0,Y 310.482,Z 1119.452,A -85,B 0,C 180,E1 21710.714,E2 21710.714} C_VEL
LIN {X 0,Y 319.105,Z 1102.914,A -85,B 0,C 180,E1 21718.35,E2 21718.35} C_VEL
LIN {X 0,Y 332.318,Z 1079.419,A -85,B 0,C 180,E1 21725.566,E2 21725.566} C_VEL
LIN {X 0,Y 347.857,Z 1050.992,A -85,B 0,C 180,E1 21731.536,E2 21731.536} C_VEL
LIN {X 0,Y 364.029,Z 1018.529,A -85,B 0,C 180,E1 21736.283,E2 21736.283} C_VEL
LIN {X 0,Y 380.004,Z 980.859,A -85,B 0,C 180,E1 21740.129,E2 21740.129} C_VEL
LIN {X 0,Y 394.317,Z 939.131,A -85,B 0,C 180,E1 21743.003,E2 21743.003} C_VEL
LIN {X 0,Y 390.023,Z 919.971,A -85,B 0,C 180,E1 21746.074,E2 21746.074} C_VEL
LIN {X 0,Y 381.012,Z 894.619,A -85,B 0,C 180,E1 21751.063,E2 21751.063} C_VEL
LIN {X 0,Y 371.159,Z 873.68,A -85,B 0,C 180,E1 21756.379,E2 21756.379} C_VEL
LIN {X 0,Y 362.027,Z 857.149,A -85,B 0,C 180,E1 21762.171,E2 21762.171} C_VEL
LIN {X 0,Y 357.184,Z 849.75,A -85,B 0,C 180,E1 21766.109,E2 21766.109} C_VEL
LIN {X 0,Y 354.161,Z 844.493,A -85,B 0,C 180,E1 21769.36,E2 21769.36} C_VEL
LIN {X 0,Y 351.102,Z 838.007,A -85,B 0,C 180,E1 21775.66,E2 21775.66} C_VEL
LIN {X 0,Y 351.399,Z 838.827,A -85,B 0,C 180,E1 21782.307,E2 21782.307} C_VEL
LIN {X 0,Y 355.473,Z 846.472,A -85,B 0,C 180,E1 21788.956,E2 21788.956} C_VEL
LIN {X 0,Y 360.123,Z 854.465,A -85,B 0,C 180,E1 21793.292,E2 21793.292} C_VEL
LIN {X 0,Y 367.617,Z 867.359,A -85,B 0,C 180,E1 21798.423,E2 21798.423} C_VEL
LIN {X 0,Y 377.311,Z 886.984,A -85,B 0,C 180,E1 21803.979,E2 21803.979} C_VEL
LIN {X 0,Y 386.433,Z 910.519,A -85,B 0,C 180,E1 21808.953,E2 21808.953} C_VEL
LIN {X 0,Y 393.527,Z 937,A -85,B 0,C 180,E1 21813.499,E2 21813.499} C_VEL
LIN {X 0,Y 393.098,Z 942.752,A -85,B 0,C 180,E1 21814.062,E2 21814.062} C_VEL
LIN {X 0,Y 379.234,Z 983.92,A -85,B 0,C 180,E1 21816.956,E2 21816.956} C_VEL
LIN {X 0,Y 362.855,Z 1023.487,A -85,B 0,C 180,E1 21820.955,E2 21820.955} C_VEL
LIN {X 0,Y 346.501,Z 1057.833,A -85,B 0,C 180,E1 21825.916,E2 21825.916} C_VEL
LIN {X 0,Y 331.402,Z 1087.163,A -85,B 0,C 180,E1 21831.884,E2 21831.884} C_VEL
LIN {X 0,Y 319.42,Z 1110.635,A -85,B 0,C 180,E1 21838.602,E2 21838.602} C_VEL
LIN {X 0,Y 310.55,Z 1129.507,A -85,B 0,C 180,E1 21846.262,E2 21846.262} C_VEL
LIN {X 0,Y 305.645,Z 1143.273,A -85,B 0,C 180,E1 21854.741,E2 21854.741} C_VEL
LIN {X 0,Y 304.287,Z 1149.677,A -85,B 0,C 180,E1 21861.406,E2 21861.406} C_VEL
LIN {X 0,Y 304.004,Z 1152.391,A -85,B 0,C 180,E1 21867.141,E2 21867.141} C_VEL
LIN {X 0,Y 304.008,Z 1152.395,A -85,B 0,C 180,E1 21872.854,E2 21872.854} C_VEL
LIN {X 0,Y 304.385,Z 1148.604,A -85,B 0,C 180,E1 21880.031,E2 21880.031} C_VEL
LIN {X 0,Y 306.807,Z 1139.584,A -85,B 0,C 180,E1 21887.976,E2 21887.976} C_VEL
LIN {X 0,Y 313.165,Z 1123.75,A -85,B 0,C 180,E1 21896.417,E2 21896.417} C_VEL
LIN {X 0,Y 323.142,Z 1103.14,A -85,B 0,C 180,E1 21903.832,E2 21903.832} C_VEL
LIN {X 0,Y 336.026,Z 1078.339,A -85,B 0,C 180,E1 21910.17,E2 21910.17} C_VEL
LIN {X 0,Y 351.618,Z 1047.728,A -85,B 0,C 180,E1 21915.754,E2 21915.754} C_VEL
LIN {X 0,Y 367.946,Z 1012.249,A -85,B 0,C 180,E1 21920.355,E2 21920.355} C_VEL
LIN {X 0,Y 384.132,Z 970.934,A -85,B 0,C 180,E1 21924.093,E2 21924.093} C_VEL
LIN {X 0,Y 394.134,Z 938.901,A -85,B 0,C 180,E1 21926.212,E2 21926.212} C_VEL
LIN {X 0,Y 386.813,Z 911.149,A -85,B 0,C 180,E1 21930.953,E2 21930.953} C_VEL
LIN {X 0,Y 376.98,Z 886.001,A -85,B 0,C 180,E1 21936.313,E2 21936.313} C_VEL
LIN {X 0,Y 367.538,Z 867.064,A -85,B 0,C 180,E1 21941.768,E2 21941.768} C_VEL
LIN {X 0,Y 360.538,Z 855.171,A -85,B 0,C 180,E1 21946.558,E2 21946.558} C_VEL
LIN {X 0,Y 357.526,Z 850.048,A -85,B 0,C 180,E1 21949.208,E2 21949.208} C_VEL
LIN {X 0,Y 357.246,Z 849.729,A -85,B 0,C 180,E1 21949.463,E2 21949.463} C_VEL
LIN {X 0,Y 353.948,Z 849.886,A -85,B 0,C 180,E1 21952.255,E2 21952.255} C_VEL
LIN {X 0,Y 351.428,Z 850.415,A -85,B 0,C 180,E1 21955.102,E2 21955.102} C_VEL
LIN {X 0,Y 350.181,Z 845.818,A -85,B 0,C 180,E1 21959.39,E2 21959.39} C_VEL
LIN {X 0,Y 350.254,Z 846.731,A -85,B 0,C 180,E1 21964.468,E2 21964.468} C_VEL
LIN {X 0,Y 353.937,Z 854.152,A -85,B 0,C 180,E1 21971.585,E2 21971.585} C_VEL
LIN {X 0,Y 358.392,Z 862.178,A -85,B 0,C 180,E1 21976.037,E2 21976.037} C_VEL
LIN {X 0,Y 365.335,Z 874.57,A -85,B 0,C 180,E1 21981.126,E2 21981.126} C_VEL
LIN {X 0,Y 374.801,Z 894.516,A -85,B 0,C 180,E1 21986.855,E2 21986.855} C_VEL
LIN {X 0,Y 383.322,Z 917.932,A -85,B 0,C 180,E1 21991.923,E2 21991.923} C_VEL
LIN {X 0,Y 389.065,Z 940.682,A -85,B 0,C 180,E1 21995.941,E2 21995.941} C_VEL
LIN {X 0,Y 375.129,Z 981.475,A -85,B 0,C 180,E1 21998.876,E2 21998.876} C_VEL
LIN {X 0,Y 359.094,Z 1017.934,A -85,B 0,C 180,E1 22002.572,E2 22002.572} C_VEL
LIN {X 0,Y 342.032,Z 1051.186,A -85,B 0,C 180,E1 22007.444,E2 22007.444} C_VEL
LIN {X 0,Y 325.599,Z 1080.132,A -85,B 0,C 180,E1 22013.61,E2 22013.61} C_VEL
LIN {X 0,Y 311.908,Z 1103.419,A -85,B 0,C 180,E1 22020.94,E2 22020.94} C_VEL
LIN {X 0,Y 302.874,Z 1120.018,A -85,B 0,C 180,E1 22028.823,E2 22028.823} C_VEL
LIN {X 0,Y 298.011,Z 1130.5,A -85,B 0,C 180,E1 22036.777,E2 22036.777} C_VEL
LIN {X 0,Y 296.347,Z 1135.744,A -85,B 0,C 180,E1 22044.133,E2 22044.133} C_VEL
LIN {X 0,Y 296.377,Z 1136.999,A -85,B 0,C 180,E1 22050.003,E2 22050.003} C_VEL
LIN {X 0,Y 296.418,Z 1135.7,A -85,B 0,C 180,E1 22055.87,E2 22055.87} C_VEL
LIN {X 0,Y 298.038,Z 1130.37,A -85,B 0,C 180,E1 22063.227,E2 22063.227} C_VEL
LIN {X 0,Y 302.926,Z 1119.789,A -85,B 0,C 180,E1 22071.184,E2 22071.184} C_VEL
LIN {X 0,Y 312.067,Z 1103.098,A -85,B 0,C 180,E1 22079.068,E2 22079.068} C_VEL
LIN {X 0,Y 325.796,Z 1079.722,A -85,B 0,C 180,E1 22086.37,E2 22086.37} C_VEL
LIN {X 0,Y 341.711,Z 1051.625,A -85,B 0,C 180,E1 22092.362,E2 22092.362} C_VEL
LIN {X 0,Y 359.135,Z 1017.641,A -85,B 0,C 180,E1 22097.342,E2 22097.342} C_VEL
LIN {X 0,Y 375.447,Z 980.029,A -85,B 0,C 180,E1 22101.152,E2 22101.152} C_VEL
LIN {X 0,Y 389.022,Z 940.875,A -85,B 0,C 180,E1 22103.902,E2 22103.902} C_VEL
LIN {X 0,Y 382.112,Z 914.491,A -85,B 0,C 180,E1 22108.632,E2 22108.632} C_VEL
LIN {X 0,Y 372.968,Z 890.602,A -85,B 0,C 180,E1 22113.978,E2 22113.978} C_VEL
LIN {X 0,Y 364.007,Z 872.267,A -85,B 0,C 180,E1 22119.511,E2 22119.511} C_VEL
LIN {X 0,Y 356.867,Z 858.89,A -85,B 0,C 180,E1 22125.076,E2 22125.076} C_VEL
LIN {X 0,Y 352.545,Z 852.018,A -85,B 0,C 180,E1 22129.78,E2 22129.78} C_VEL
LIN {X 0,Y 349.815,Z 845.747,A -85,B 0,C 180,E1 22136.266,E2 22136.266} C_VEL
LIN {X 0,Y 350.196,Z 846.621,A -85,B 0,C 180,E1 22142.16,E2 22142.16} C_VEL
LIN {X 0,Y 353.929,Z 854.308,A -85,B 0,C 180,E1 22148.84,E2 22148.84} C_VEL
LIN {X 0,Y 358.341,Z 862.233,A -85,B 0,C 180,E1 22153.155,E2 22153.155} C_VEL
LIN {X 0,Y 366.08,Z 876.443,A -85,B 0,C 180,E1 22158.761,E2 22158.761} C_VEL
LIN {X 0,Y 374.939,Z 895.941,A -85,B 0,C 180,E1 22164.14,E2 22164.14} C_VEL
LIN {X 0,Y 383.393,Z 920.701,A -85,B 0,C 180,E1 22169.331,E2 22169.331} C_VEL
LIN {X 0,Y 388.543,Z 942.448,A -85,B 0,C 180,E1 22173.076,E2 22173.076} C_VEL
LIN {X 0,Y 373.869,Z 985.078,A -85,B 0,C 180,E1 22176.096,E2 22176.096} C_VEL
LIN {X 0,Y 356.891,Z 1024.745,A -85,B 0,C 180,E1 22180.163,E2 22180.163} C_VEL
LIN {X 0,Y 339.527,Z 1059.856,A -85,B 0,C 180,E1 22185.349,E2 22185.349} C_VEL
LIN {X 0,Y 323.666,Z 1089.632,A -85,B 0,C 180,E1 22191.661,E2 22191.661} C_VEL
LIN {X 0,Y 310.311,Z 1114.632,A -85,B 0,C 180,E1 22199.304,E2 22199.304} C_VEL
LIN {X 0,Y 301.682,Z 1132.49,A -85,B 0,C 180,E1 22207.341,E2 22207.341} C_VEL
LIN {X 0,Y 297.564,Z 1144.098,A -85,B 0,C 180,E1 22215.28,E2 22215.28} C_VEL
LIN {X 0,Y 296.397,Z 1149.467,A -85,B 0,C 180,E1 22221.176,E2 22221.176} C_VEL
LIN {X 0,Y 296.101,Z 1152.183,A -85,B 0,C 180,E1 22227.064,E2 22227.064} C_VEL
LIN {X 0,Y 296.104,Z 1152.188,A -85,B 0,C 180,E1 22232.931,E2 22232.931} C_VEL
LIN {X 0,Y 296.539,Z 1148.394,A -85,B 0,C 180,E1 22240.299,E2 22240.299} C_VEL
LIN {X 0,Y 299.104,Z 1139.37,A -85,B 0,C 180,E1 22248.455,E2 22248.455} C_VEL
LIN {X 0,Y 305.61,Z 1124.058,A -85,B 0,C 180,E1 22256.856,E2 22256.856} C_VEL
LIN {X 0,Y 315.775,Z 1104.02,A -85,B 0,C 180,E1 22264.315,E2 22264.315} C_VEL
LIN {X 0,Y 329.409,Z 1078.877,A -85,B 0,C 180,E1 22270.918,E2 22270.918} C_VEL
LIN {X 0,Y 345.974,Z 1047.452,A -85,B 0,C 180,E1 22276.722,E2 22276.722} C_VEL
LIN {X 0,Y 363.23,Z 1010.992,A -85,B 0,C 180,E1 22281.444,E2 22281.444} C_VEL
LIN {X 0,Y 379.118,Z 971.479,A -85,B 0,C 180,E1 22285.01,E2 22285.01} C_VEL
LIN {X 0,Y 388.729,Z 942.396,A -85,B 0,C 180,E1 22286.942,E2 22286.942} C_VEL
LIN {X 0,Y 382.131,Z 915.976,A -85,B 0,C 180,E1 22291.601,E2 22291.601} C_VEL
LIN {X 0,Y 372.779,Z 890.613,A -85,B 0,C 180,E1 22297.219,E2 22297.219} C_VEL
LIN {X 0,Y 363.499,Z 871.166,A -85,B 0,C 180,E1 22303.125,E2 22303.125} C_VEL
LIN {X 0,Y 356.195,Z 858.162,A -85,B 0,C 180,E1 22309.006,E2 22309.006} C_VEL
LIN {X 0,Y 352.742,Z 852.047,A -85,B 0,C 180,E1 22313.071,E2 22313.071} C_VEL
LIN {X 0,Y 351.428,Z 850.415,A -85,B 0,C 180,E1 22315.102,E2 22315.102} C_VEL
LIN {X 0,Y 349.733,Z 851.269,A -85,B 0,C 180,E1 22317.96,E2 22317.96} C_VEL
LIN {X 0,Y 348.649,Z 853.499,A -85,B 0,C 180,E1 22320.856,E2 22320.856} C_VEL
LIN {X 0,Y 348.848,Z 854.648,A -85,B 0,C 180,E1 22324.414,E2 22324.414} C_VEL
LIN {X 0,Y 352.185,Z 861.734,A -85,B 0,C 180,E1 22331.328,E2 22331.328} C_VEL
LIN {X 0,Y 356.669,Z 870.344,A -85,B 0,C 180,E1 22336.116,E2 22336.116} C_VEL
LIN {X 0,Y 363.458,Z 883.262,A -85,B 0,C 180,E1 22341.32,E2 22341.32} C_VEL
LIN {X 0,Y 371.54,Z 901.919,A -85,B 0,C 180,E1 22346.66,E2 22346.66} C_VEL
LIN {X 0,Y 379.088,Z 924.274,A -85,B 0,C 180,E1 22351.565,E2 22351.565} C_VEL
LIN {X 0,Y 383.5,Z 945.139,A -85,B 0,C 180,E1 22355.307,E2 22355.307} C_VEL
LIN {X 0,Y 369.542,Z 983.335,A -85,B 0,C 180,E1 22358.054,E2 22358.054} C_VEL
LIN {X 0,Y 353.761,Z 1018.226,A -85,B 0,C 180,E1 22361.623,E2 22361.623} C_VEL
LIN {X 0,Y 335.867,Z 1051.967,A -85,B 0,C 180,E1 22366.61,E2 22366.61} C_VEL
LIN {X 0,Y 319.133,Z 1080.364,A -85,B 0,C 180,E1 22372.75,E2 22372.75} C_VEL
LIN {X 0,Y 304.888,Z 1103.637,A -85,B 0,C 180,E1 22380.204,E2 22380.204} C_VEL
LIN {X 0,Y 295.712,Z 1119.573,A -85,B 0,C 180,E1 22387.882,E2 22387.882} C_VEL
LIN {X 0,Y 290.26,Z 1130.71,A -85,B 0,C 180,E1 22396.417,E2 22396.417} C_VEL
LIN {X 0,Y 288.491,Z 1135.951,A -85,B 0,C 180,E1 22403.973,E2 22403.973} C_VEL
LIN {X 0,Y 288.475,Z 1137.206,A -85,B 0,C 180,E1 22410.003,E2 22410.003} C_VEL
LIN {X 0,Y 288.545,Z 1135.907,A -85,B 0,C 180,E1 22416.031,E2 22416.031} C_VEL
LIN {X 0,Y 290.287,Z 1130.582,A -85,B 0,C 180,E1 22423.587,E2 22423.587} C_VEL
LIN {X 0,Y 295.758,Z 1119.334,A -85,B 0,C 180,E1 22432.134,E2 22432.134} C_VEL
LIN {X 0,Y 305.013,Z 1103.361,A -85,B 0,C 180,E1 22439.788,E2 22439.788} C_VEL
LIN {X 0,Y 319.356,Z 1079.961,A -85,B 0,C 180,E1 22447.226,E2 22447.226} C_VEL
LIN {X 0,Y 336.276,Z 1051.068,A -85,B 0,C 180,E1 22453.425,E2 22453.425} C_VEL
LIN {X 0,Y 354.091,Z 1017.287,A -85,B 0,C 180,E1 22458.368,E2 22458.368} C_VEL
LIN {X 0,Y 370.502,Z 980.442,A -85,B 0,C 180,E1 22462.105,E2 22462.105} C_VEL
LIN {X 0,Y 383.585,Z 944.405,A -85,B 0,C 180,E1 22464.627,E2 22464.627} C_VEL
LIN {X 0,Y 377.154,Z 918.222,A -85,B 0,C 180,E1 22469.516,E2 22469.516} C_VEL
LIN {X 0,Y 368.719,Z 895.175,A -85,B 0,C 180,E1 22474.955,E2 22474.955} C_VEL
LIN {X 0,Y 360.067,Z 876.608,A -85,B 0,C 180,E1 22480.879,E2 22480.879} C_VEL
LIN {X 0,Y 353.985,Z 865.355,A -85,B 0,C 180,E1 22486.218,E2 22486.218} C_VEL
LIN {X 0,Y 350.828,Z 859.626,A -85,B 0,C 180,E1 22490.044,E2 22490.044} C_VEL
LIN {X 0,Y 348.499,Z 853.537,A -85,B 0,C 180,E1 22496.252,E2 22496.252} C_VEL
LIN {X 0,Y 348.769,Z 854.326,A -85,B 0,C 180,E1 22501.982,E2 22501.982} C_VEL
LIN {X 0,Y 352.149,Z 861.86,A -85,B 0,C 180,E1 22508.573,E2 22508.573} C_VEL
LIN {X 0,Y 356.711,Z 870.563,A -85,B 0,C 180,E1 22513.343,E2 22513.343} C_VEL
LIN {X 0,Y 363.624,Z 884.419,A -85,B 0,C 180,E1 22518.671,E2 22518.671} C_VEL
LIN {X 0,Y 371.277,Z 902.544,A -85,B 0,C 180,E1 22523.754,E2 22523.754} C_VEL
LIN {X 0,Y 379.169,Z 927.349,A -85,B 0,C 180,E1 22529.033,E2 22529.033} C_VEL
LIN {X 0,Y 382.869,Z 946.354,A -85,B 0,C 180,E1 22532.352,E2 22532.352} C_VEL
LIN {X 0,Y 368.396,Z 986.539,A -85,B 0,C 180,E1 22535.239,E2 22535.239} C_VEL
LIN {X 0,Y 351.155,Z 1025.521,A -85,B 0,C 180,E1 22539.285,E2 22539.285} C_VEL
LIN {X 0,Y 333.782,Z 1059.589,A -85,B 0,C 180,E1 22544.366,E2 22544.366} C_VEL
LIN {X 0,Y 317.092,Z 1089.599,A -85,B 0,C 180,E1 22550.786,E2 22550.786} C_VEL
LIN {X 0,Y 303.64,Z 1113.718,A -85,B 0,C 180,E1 22558.267,E2 22558.267} C_VEL
LIN {X 0,Y 294.377,Z 1131.827,A -85,B 0,C 180,E1 22566.489,E2 22566.489} C_VEL
LIN {X 0,Y 289.78,Z 1143.85,A -85,B 0,C 180,E1 22574.842,E2 22574.842} C_VEL
LIN {X 0,Y 288.514,Z 1149.257,A -85,B 0,C 180,E1 22580.933,E2 22580.933} C_VEL
LIN {X 0,Y 288.197,Z 1151.976,A -85,B 0,C 180,E1 22586.984,E2 22586.984} C_VEL
LIN {X 0,Y 288.195,Z 1151.98,A -85,B 0,C 180,E1 22593.011,E2 22593.011} C_VEL
LIN {X 0,Y 288.676,Z 1148.183,A -85,B 0,C 180,E1 22600.583,E2 22600.583} C_VEL
LIN {X 0,Y 291.422,Z 1139.155,A -85,B 0,C 180,E1 22608.96,E2 22608.96} C_VEL
LIN {X 0,Y 297.988,Z 1124.551,A -85,B 0,C 180,E1 22617.231,E2 22617.231} C_VEL
LIN {X 0,Y 308.448,Z 1104.9,A -85,B 0,C 180,E1 22624.82,E2 22624.82} C_VEL
LIN {X 0,Y 322.546,Z 1080.006,A -85,B 0,C 180,E1 22631.566,E2 22631.566} C_VEL
LIN {X 0,Y 339.416,Z 1049.144,A -85,B 0,C 180,E1 22637.415,E2 22637.415} C_VEL
LIN {X 0,Y 357.557,Z 1012.2,A -85,B 0,C 180,E1 22642.292,E2 22642.292} C_VEL
LIN {X 0,Y 374.55,Z 971.107,A -85,B 0,C 180,E1 22646.021,E2 22646.021} C_VEL
LIN {X 0,Y 383.189,Z 945.313,A -85,B 0,C 180,E1 22647.769,E2 22647.769} C_VEL
LIN {X 0,Y 377.104,Z 919.755,A -85,B 0,C 180,E1 22652.491,E2 22652.491} C_VEL
LIN {X 0,Y 369.311,Z 896.963,A -85,B 0,C 180,E1 22657.709,E2 22657.709} C_VEL
LIN {X 0,Y 360.632,Z 877.636,A -85,B 0,C 180,E1 22663.719,E2 22663.719} C_VEL
LIN {X 0,Y 353.888,Z 865.127,A -85,B 0,C 180,E1 22669.694,E2 22669.694} C_VEL
LIN {X 0,Y 351.021,Z 859.588,A -85,B 0,C 180,E1 22673.348,E2 22673.348} C_VEL
LIN {X 0,Y 348.748,Z 853.494,A -85,B 0,C 180,E1 22680.009,E2 22680.009} C_VEL
LIN {X 0,Y 348.649,Z 853.499,A -85,B 0,C 180,E1 22680.856,E2 22680.856} C_VEL
LIN {X 0,Y 348.152,Z 856.53,A -85,B 0,C 180,E1 22682.955,E2 22682.955} C_VEL
LIN {X 0,Y 347.699,Z 864.783,A -85,B 0,C 180,E1 22686.372,E2 22686.372} C_VEL
LIN {X 0,Y 350.27,Z 869.268,A -85,B 0,C 180,E1 22691.075,E2 22691.075} C_VEL
LIN {X 0,Y 355.744,Z 879.748,A -85,B 0,C 180,E1 22696.955,E2 22696.955} C_VEL
LIN {X 0,Y 362.955,Z 895.769,A -85,B 0,C 180,E1 22702.723,E2 22702.723} C_VEL
LIN {X 0,Y 370.882,Z 917.114,A -85,B 0,C 180,E1 22708.361,E2 22708.361} C_VEL
LIN {X 0,Y 377.303,Z 942.228,A -85,B 0,C 180,E1 22713.46,E2 22713.46} C_VEL
LIN {X 0,Y 378.209,Z 947.703,A -85,B 0,C 180,E1 22714.446,E2 22714.446} C_VEL
LIN {X 0,Y 364.221,Z 984.802,A -85,B 0,C 180,E1 22717.175,E2 22717.175} C_VEL
LIN {X 0,Y 347.825,Z 1019.823,A -85,B 0,C 180,E1 22720.807,E2 22720.807} C_VEL
LIN {X 0,Y 330.256,Z 1051.901,A -85,B 0,C 180,E1 22725.594,E2 22725.594} C_VEL
LIN {X 0,Y 312.78,Z 1080.594,A -85,B 0,C 180,E1 22731.86,E2 22731.86} C_VEL
LIN {X 0,Y 297.939,Z 1103.854,A -85,B 0,C 180,E1 22739.436,E2 22739.436} C_VEL
LIN {X 0,Y 288.164,Z 1120.015,A -85,B 0,C 180,E1 22747.413,E2 22747.413} C_VEL
LIN {X 0,Y 282.514,Z 1130.919,A -85,B 0,C 180,E1 22756.037,E2 22756.037} C_VEL
LIN {X 0,Y 280.605,Z 1136.159,A -85,B 0,C 180,E1 22763.803,E2 22763.803} C_VEL
LIN {X 0,Y 280.581,Z 1137.413,A -85,B 0,C 180,E1 22770.003,E2 22770.003} C_VEL
LIN {X 0,Y 280.656,Z 1136.115,A -85,B 0,C 180,E1 22776.201,E2 22776.201} C_VEL
LIN {X 0,Y 282.541,Z 1130.794,A -85,B 0,C 180,E1 22783.967,E2 22783.967} C_VEL
LIN {X 0,Y 288.21,Z 1119.78,A -85,B 0,C 180,E1 22792.601,E2 22792.601} C_VEL
LIN {X 0,Y 298.066,Z 1103.583,A -85,B 0,C 180,E1 22800.556,E2 22800.556} C_VEL
LIN {X 0,Y 312.966,Z 1080.201,A -85,B 0,C 180,E1 22808.12,E2 22808.12} C_VEL
LIN {X 0,Y 329.642,Z 1052.793,A -85,B 0,C 180,E1 22814.115,E2 22814.115} C_VEL
LIN {X 0,Y 347.732,Z 1019.786,A -85,B 0,C 180,E1 22819.077,E2 22819.077} C_VEL
LIN {X 0,Y 365.076,Z 982.244,A -85,B 0,C 180,E1 22822.961,E2 22822.961} C_VEL
LIN {X 0,Y 378.063,Z 947.154,A -85,B 0,C 180,E1 22825.516,E2 22825.516} C_VEL
LIN {X 0,Y 372.273,Z 922.13,A -85,B 0,C 180,E1 22830.405,E2 22830.405} C_VEL
LIN {X 0,Y 364.625,Z 900.234,A -85,B 0,C 180,E1 22835.798,E2 22835.798} C_VEL
LIN {X 0,Y 357.094,Z 883.011,A -85,B 0,C 180,E1 22841.533,E2 22841.533} C_VEL
LIN {X 0,Y 351.71,Z 872.645,A -85,B 0,C 180,E1 22846.603,E2 22846.603} C_VEL
LIN {X 0,Y 349.039,Z 867.201,A -85,B 0,C 180,E1 22850.308,E2 22850.308} C_VEL
LIN {X 0,Y 347.013,Z 861.273,A -85,B 0,C 180,E1 22856.236,E2 22856.236} C_VEL
LIN {X 0,Y 347.22,Z 862.01,A -85,B 0,C 180,E1 22861.803,E2 22861.803} C_VEL
LIN {X 0,Y 350.229,Z 869.513,A -85,B 0,C 180,E1 22868.386,E2 22868.386} C_VEL
LIN {X 0,Y 354.92,Z 878.731,A -85,B 0,C 180,E1 22873.49,E2 22873.49} C_VEL
LIN {X 0,Y 362.059,Z 894.392,A -85,B 0,C 180,E1 22879.31,E2 22879.31} C_VEL
LIN {X 0,Y 369.264,Z 914.003,A -85,B 0,C 180,E1 22884.536,E2 22884.536} C_VEL
LIN {X 0,Y 375.712,Z 938.319,A -85,B 0,C 180,E1 22889.592,E2 22889.592} C_VEL
LIN {X 0,Y 377.4,Z 949.59,A -85,B 0,C 180,E1 22891.548,E2 22891.548} C_VEL
LIN {X 0,Y 363.286,Z 987.399,A -85,B 0,C 180,E1 22894.31,E2 22894.31} C_VEL
LIN {X 0,Y 346.048,Z 1025.23,A -85,B 0,C 180,E1 22898.24,E2 22898.24} C_VEL
LIN {X 0,Y 327.921,Z 1059.683,A -85,B 0,C 180,E1 22903.411,E2 22903.411} C_VEL
LIN {X 0,Y 310.648,Z 1089.567,A -85,B 0,C 180,E1 22909.883,E2 22909.883} C_VEL
LIN {X 0,Y 296.465,Z 1113.959,A -85,B 0,C 180,E1 22917.611,E2 22917.611} C_VEL
LIN {X 0,Y 286.307,Z 1132.985,A -85,B 0,C 180,E1 22926.612,E2 22926.612} C_VEL
LIN {X 0,Y 281.702,Z 1144.694,A -85,B 0,C 180,E1 22935.434,E2 22935.434} C_VEL
LIN {X 0,Y 280.318,Z 1150.739,A -85,B 0,C 180,E1 22943.791,E2 22943.791} C_VEL
LIN {X 0,Y 280.505,Z 1152.128,A -85,B 0,C 180,E1 22949.997,E2 22949.997} C_VEL
LIN {X 0,Y 280.307,Z 1150.751,A -85,B 0,C 180,E1 22956.204,E2 22956.204} C_VEL
LIN {X 0,Y 281.708,Z 1144.721,A -85,B 0,C 180,E1 22964.571,E2 22964.571} C_VEL
LIN {X 0,Y 286.302,Z 1133.054,A -85,B 0,C 180,E1 22973.382,E2 22973.382} C_VEL
LIN {X 0,Y 296.378,Z 1114.113,A -85,B 0,C 180,E1 22982.369,E2 22982.369} C_VEL
LIN {X 0,Y 310.562,Z 1089.731,A -85,B 0,C 180,E1 22990.114,E2 22990.114} C_VEL
LIN {X 0,Y 327.89,Z 1059.891,A -85,B 0,C 180,E1 22996.582,E2 22996.582} C_VEL
LIN {X 0,Y 346.668,Z 1024.413,A -85,B 0,C 180,E1 23001.876,E2 23001.876} C_VEL
LIN {X 0,Y 364.009,Z 986.161,A -85,B 0,C 180,E1 23005.815,E2 23005.815} C_VEL
LIN {X 0,Y 377.738,Z 948.483,A -85,B 0,C 180,E1 23008.584,E2 23008.584} C_VEL
LIN {X 0,Y 372.195,Z 923.443,A -85,B 0,C 180,E1 23013.41,E2 23013.41} C_VEL
LIN {X 0,Y 364.915,Z 901.405,A -85,B 0,C 180,E1 23018.708,E2 23018.708} C_VEL
LIN {X 0,Y 357.483,Z 884.019,A -85,B 0,C 180,E1 23024.414,E2 23024.414} C_VEL
LIN {X 0,Y 351.758,Z 872.583,A -85,B 0,C 180,E1 23029.932,E2 23029.932} C_VEL
LIN {X 0,Y 349.205,Z 867.165,A -85,B 0,C 180,E1 23033.626,E2 23033.626} C_VEL
LIN {X 0,Y 347.26,Z 861.226,A -85,B 0,C 180,E1 23040.009,E2 23040.009} C_VEL
LIN {X 0,Y 347.315,Z 862.325,A -85,B 0,C 180,E1 23044.231,E2 23044.231} C_VEL
LIN {X 0,Y 347.699,Z 864.783,A -85,B 0,C 180,E1 23046.372,E2 23046.372} C_VEL
LIN {X 0,Y 347.991,Z 871.195,A -85,B 0,C 180,E1 23049.075,E2 23049.075} C_VEL
LIN {X 0,Y 348.771,Z 878.379,A -85,B 0,C 180,E1 23051.744,E2 23051.744} C_VEL
LIN {X 0,Y 353.114,Z 886.973,A -85,B 0,C 180,E1 23056.636,E2 23056.636} C_VEL
LIN {X 0,Y 360.113,Z 903.819,A -85,B 0,C 180,E1 23062.74,E2 23062.74} C_VEL
LIN {X 0,Y 367.505,Z 925.64,A -85,B 0,C 180,E1 23068.465,E2 23068.465} C_VEL
LIN {X 0,Y 372.755,Z 950.226,A -85,B 0,C 180,E1 23073.493,E2 23073.493} C_VEL
LIN {X 0,Y 358.734,Z 986.824,A -85,B 0,C 180,E1 23076.318,E2 23076.318} C_VEL
LIN {X 0,Y 342.679,Z 1020.099,A -85,B 0,C 180,E1 23079.8,E2 23079.8} C_VEL
LIN {X 0,Y 323.739,Z 1053.492,A -85,B 0,C 180,E1 23084.856,E2 23084.856} C_VEL
LIN {X 0,Y 306.492,Z 1080.823,A -85,B 0,C 180,E1 23090.931,E2 23090.931} C_VEL
LIN {X 0,Y 291.027,Z 1104.072,A -85,B 0,C 180,E1 23098.629,E2 23098.629} C_VEL
LIN {X 0,Y 280.486,Z 1120.713,A -85,B 0,C 180,E1 23107.071,E2 23107.071} C_VEL
LIN {X 0,Y 274.731,Z 1131.213,A -85,B 0,C 180,E1 23115.723,E2 23115.723} C_VEL
LIN {X 0,Y 272.735,Z 1136.366,A -85,B 0,C 180,E1 23123.624,E2 23123.624} C_VEL
LIN {X 0,Y 272.696,Z 1137.62,A -85,B 0,C 180,E1 23130.003,E2 23130.003} C_VEL
LIN {X 0,Y 272.778,Z 1136.323,A -85,B 0,C 180,E1 23136.381,E2 23136.381} C_VEL
LIN {X 0,Y 274.768,Z 1131.074,A -85,B 0,C 180,E1 23144.296,E2 23144.296} C_VEL
LIN {X 0,Y 280.521,Z 1120.497,A -85,B 0,C 180,E1 23152.934,E2 23152.934} C_VEL
LIN {X 0,Y 291.143,Z 1103.805,A -85,B 0,C 180,E1 23161.363,E2 23161.363} C_VEL
LIN {X 0,Y 306.662,Z 1080.438,A -85,B 0,C 180,E1 23169.05,E2 23169.05} C_VEL
LIN {X 0,Y 324.642,Z 1051.875,A -85,B 0,C 180,E1 23175.322,E2 23175.322} C_VEL
LIN {X 0,Y 343.653,Z 1018.021,A -85,B 0,C 180,E1 23180.337,E2 23180.337} C_VEL
LIN {X 0,Y 360.987,Z 981.19,A -85,B 0,C 180,E1 23184.085,E2 23184.085} C_VEL
LIN {X 0,Y 372.644,Z 950.207,A -85,B 0,C 180,E1 23186.384,E2 23186.384} C_VEL
LIN {X 0,Y 367.369,Z 925.758,A -85,B 0,C 180,E1 23191.387,E2 23191.387} C_VEL
LIN {X 0,Y 360.208,Z 904.379,A -85,B 0,C 180,E1 23196.932,E2 23196.932} C_VEL
LIN {X 0,Y 352.964,Z 886.698,A -85,B 0,C 180,E1 23203.229,E2 23203.229} C_VEL
LIN {X 0,Y 348.423,Z 877.828,A -85,B 0,C 180,E1 23208.309,E2 23208.309} C_VEL
LIN {X 0,Y 346.811,Z 874.447,A -85,B 0,C 180,E1 23210.879,E2 23210.879} C_VEL
LIN {X 0,Y 345.362,Z 868.972,A -85,B 0,C 180,E1 23216.218,E2 23216.218} C_VEL
LIN {X 0,Y 345.478,Z 869.758,A -85,B 0,C 180,E1 23221.718,E2 23221.718} C_VEL
LIN {X 0,Y 348.181,Z 877.1,A -85,B 0,C 180,E1 23228.199,E2 23228.199} C_VEL
LIN {X 0,Y 352.692,Z 886.546,A -85,B 0,C 180,E1 23233.498,E2 23233.498} C_VEL
LIN {X 0,Y 359.297,Z 902.769,A -85,B 0,C 180,E1 23239.384,E2 23239.384} C_VEL
LIN {X 0,Y 365.68,Z 921.756,A -85,B 0,C 180,E1 23244.466,E2 23244.466} C_VEL
LIN {X 0,Y 371.333,Z 946.305,A -85,B 0,C 180,E1 23249.601,E2 23249.601} C_VEL
LIN {X 0,Y 372.209,Z 952.249,A -85,B 0,C 180,E1 23250.687,E2 23250.687} C_VEL
LIN {X 0,Y 357.399,Z 990.191,A -85,B 0,C 180,E1 23253.519,E2 23253.519} C_VEL
LIN {X 0,Y 339.972,Z 1027.073,A -85,B 0,C 180,E1 23257.449,E2 23257.449} C_VEL
LIN {X 0,Y 321.956,Z 1060.106,A -85,B 0,C 180,E1 23262.485,E2 23262.485} C_VEL
LIN {X 0,Y 304.162,Z 1089.766,A -85,B 0,C 180,E1 23269.007,E2 23269.007} C_VEL
LIN {X 0,Y 289.447,Z 1114.016,A -85,B 0,C 180,E1 23276.854,E2 23276.854} C_VEL
LIN {X 0,Y 278.864,Z 1132.765,A -85,B 0,C 180,E1 23285.949,E2 23285.949} C_VEL
LIN {X 0,Y 273.913,Z 1144.48,A -85,B 0,C 180,E1 23295.01,E2 23295.01} C_VEL
LIN {X 0,Y 272.433,Z 1150.53,A -85,B 0,C 180,E1 23303.611,E2 23303.611} C_VEL
LIN {X 0,Y 272.61,Z 1151.921,A -85,B 0,C 180,E1 23309.997,E2 23309.997} C_VEL
LIN {X 0,Y 272.422,Z 1150.544,A -85,B 0,C 180,E1 23316.384,E2 23316.384} C_VEL
LIN {X 0,Y 273.832,Z 1144.812,A -85,B 0,C 180,E1 23324.695,E2 23324.695} C_VEL
LIN {X 0,Y 278.211,Z 1134.085,A -85,B 0,C 180,E1 23333.253,E2 23333.253} C_VEL
LIN {X 0,Y 287.46,Z 1117.323,A -85,B 0,C 180,E1 23341.806,E2 23341.806} C_VEL
LIN {X 0,Y 300.903,Z 1095.239,A -85,B 0,C 180,E1 23349.47,E2 23349.47} C_VEL
LIN {X 0,Y 317.416,Z 1067.92,A -85,B 0,C 180,E1 23356.054,E2 23356.054} C_VEL
LIN {X 0,Y 336.136,Z 1034.797,A -85,B 0,C 180,E1 23361.55,E2 23361.55} C_VEL
LIN {X 0,Y 354.331,Z 997.769,A -85,B 0,C 180,E1 23365.806,E2 23365.806} C_VEL
LIN {X 0,Y 370.917,Z 956.549,A -85,B 0,C 180,E1 23369.07,E2 23369.07} C_VEL
LIN {X 0,Y 372.252,Z 950.766,A -85,B 0,C 180,E1 23369.578,E2 23369.578} C_VEL
LIN {X 0,Y 367.295,Z 926.945,A -85,B 0,C 180,E1 23374.402,E2 23374.402} C_VEL
LIN {X 0,Y 360.7,Z 905.965,A -85,B 0,C 180,E1 23379.688,E2 23379.688} C_VEL
LIN {X 0,Y 354.254,Z 890.219,A -85,B 0,C 180,E1 23385.141,E2 23385.141} C_VEL
LIN {X 0,Y 349.475,Z 879.854,A -85,B 0,C 180,E1 23390.339,E2 23390.339} C_VEL
LIN {X 0,Y 347.068,Z 874.524,A -85,B 0,C 180,E1 23394.059,E2 23394.059} C_VEL
LIN {X 0,Y 345.593,Z 868.953,A -85,B 0,C 180,E1 23400.009,E2 23400.009} C_VEL
LIN {X 0,Y 345.574,Z 870.013,A -85,B 0,C 180,E1 23404.095,E2 23404.095} C_VEL
LIN {X 0,Y 348.287,Z 877.049,A -85,B 0,C 180,E1 23410.98,E2 23410.98} C_VEL
LIN {X 0,Y 348.771,Z 878.379,A -85,B 0,C 180,E1 23411.744,E2 23411.744} C_VEL
LIN {X 0,Y 349.675,Z 886.487,A -85,B 0,C 180,E1 23414.288,E2 23414.288} C_VEL
LIN {X 0,Y 350.878,Z 895.324,A -85,B 0,C 180,E1 23416.785,E2 23416.785} C_VEL
LIN {X 0,Y 357.242,Z 911.899,A -85,B 0,C 180,E1 23422.777,E2 23422.777} C_VEL
LIN {X 0,Y 363.456,Z 932.873,A -85,B 0,C 180,E1 23428.315,E2 23428.315} C_VEL
LIN {X 0,Y 367.556,Z 954.404,A -85,B 0,C 180,E1 23432.804,E2 23432.804} C_VEL
LIN {X 0,Y 350.786,Z 994.366,A -85,B 0,C 180,E1 23435.92,E2 23435.92} C_VEL
LIN {X 0,Y 331.956,Z 1030.758,A -85,B 0,C 180,E1 23440.138,E2 23440.138} C_VEL
LIN {X 0,Y 313.077,Z 1061.896,A -85,B 0,C 180,E1 23445.437,E2 23445.437} C_VEL
LIN {X 0,Y 294.602,Z 1089.303,A -85,B 0,C 180,E1 23452.37,E2 23452.37} C_VEL
LIN {X 0,Y 280.507,Z 1109.59,A -85,B 0,C 180,E1 23460.136,E2 23460.136} C_VEL
LIN {X 0,Y 270.424,Z 1125.243,A -85,B 0,C 180,E1 23469.505,E2 23469.505} C_VEL
LIN {X 0,Y 265.875,Z 1133.907,A -85,B 0,C 180,E1 23478.498,E2 23478.498} C_VEL
LIN {X 0,Y 264.663,Z 1137.519,A -85,B 0,C 180,E1 23486.721,E2 23486.721} C_VEL
LIN {X 0,Y 264.694,Z 1137.503,A -85,B 0,C 180,E1 23493.284,E2 23493.284} C_VEL
LIN {X 0,Y 265.896,Z 1133.81,A -85,B 0,C 180,E1 23501.507,E2 23501.507} C_VEL
LIN {X 0,Y 270.499,Z 1125.062,A -85,B 0,C 180,E1 23510.495,E2 23510.495} C_VEL
LIN {X 0,Y 279.685,Z 1110.739,A -85,B 0,C 180,E1 23519.184,E2 23519.184} C_VEL
LIN {X 0,Y 294.154,Z 1089.839,A -85,B 0,C 180,E1 23527.325,E2 23527.325} C_VEL
LIN {X 0,Y 312.268,Z 1062.924,A -85,B 0,C 180,E1 23534.23,E2 23534.23} C_VEL
LIN {X 0,Y 331.027,Z 1032.08,A -85,B 0,C 180,E1 23539.552,E2 23539.552} C_VEL
LIN {X 0,Y 349.119,Z 997.37,A -85,B 0,C 180,E1 23543.672,E2 23543.672} C_VEL
LIN {X 0,Y 365.05,Z 960.456,A -85,B 0,C 180,E1 23546.674,E2 23546.674} C_VEL
LIN {X 0,Y 367.363,Z 953.569,A -85,B 0,C 180,E1 23547.219,E2 23547.219} C_VEL
LIN {X 0,Y 362.636,Z 930.18,A -85,B 0,C 180,E1 23552.188,E2 23552.188} C_VEL
LIN {X 0,Y 356.116,Z 909.093,A -85,B 0,C 180,E1 23557.927,E2 23557.927} C_VEL
LIN {X 0,Y 349.977,Z 893.388,A -85,B 0,C 180,E1 23563.84,E2 23563.84} C_VEL
LIN {X 0,Y 345.545,Z 882.804,A -85,B 0,C 180,E1 23569.89,E2 23569.89} C_VEL
LIN {X 0,Y 343.523,Z 876.659,A -85,B 0,C 180,E1 23576.197,E2 23576.197} C_VEL
LIN {X 0,Y 343.582,Z 877.335,A -85,B 0,C 180,E1 23581.491,E2 23581.491} C_VEL
LIN {X 0,Y 345.97,Z 884.611,A -85,B 0,C 180,E1 23588.014,E2 23588.014} C_VEL
LIN {X 0,Y 350.1,Z 894.027,A -85,B 0,C 180,E1 23593.281,E2 23593.281} C_VEL
LIN {X 0,Y 356.19,Z 910.208,A -85,B 0,C 180,E1 23599.212,E2 23599.212} C_VEL
LIN {X 0,Y 361.856,Z 928.976,A -85,B 0,C 180,E1 23604.282,E2 23604.282} C_VEL
LIN {X 0,Y 366.243,Z 950.691,A -85,B 0,C 180,E1 23608.939,E2 23608.939} C_VEL
LIN {X 0,Y 366.84,Z 955.639,A -85,B 0,C 180,E1 23609.842,E2 23609.842} C_VEL
LIN {X 0,Y 350.55,Z 995.462,A -85,B 0,C 180,E1 23612.943,E2 23612.943} C_VEL
LIN {X 0,Y 332.821,Z 1031.05,A -85,B 0,C 180,E1 23616.911,E2 23616.911} C_VEL
LIN {X 0,Y 315.214,Z 1061.934,A -85,B 0,C 180,E1 23621.794,E2 23621.794} C_VEL
LIN {X 0,Y 297.909,Z 1089.726,A -85,B 0,C 180,E1 23628.03,E2 23628.03} C_VEL
LIN {X 0,Y 282.664,Z 1113.787,A -85,B 0,C 180,E1 23635.951,E2 23635.951} C_VEL
LIN {X 0,Y 271.457,Z 1132.544,A -85,B 0,C 180,E1 23645.25,E2 23645.25} C_VEL
LIN {X 0,Y 266.091,Z 1144.431,A -85,B 0,C 180,E1 23654.73,E2 23654.73} C_VEL
LIN {X 0,Y 264.53,Z 1150.322,A -85,B 0,C 180,E1 23663.419,E2 23663.419} C_VEL
LIN {X 0,Y 264.706,Z 1151.714,A -85,B 0,C 180,E1 23669.997,E2 23669.997} C_VEL
LIN {X 0,Y 264.517,Z 1150.335,A -85,B 0,C 180,E1 23676.575,E2 23676.575} C_VEL
LIN {X 0,Y 266.098,Z 1144.464,A -85,B 0,C 180,E1 23685.273,E2 23685.273} C_VEL
LIN {X 0,Y 271.452,Z 1132.618,A -85,B 0,C 180,E1 23694.745,E2 23694.745} C_VEL
LIN {X 0,Y 282.516,Z 1113.99,A -85,B 0,C 180,E1 23704.015,E2 23704.015} C_VEL
LIN {X 0,Y 297.855,Z 1089.898,A -85,B 0,C 180,E1 23711.958,E2 23711.958} C_VEL
LIN {X 0,Y 317.019,Z 1059.244,A -85,B 0,C 180,E1 23718.743,E2 23718.743} C_VEL
LIN {X 0,Y 336.89,Z 1023.828,A -85,B 0,C 180,E1 23724.048,E2 23724.048} C_VEL
LIN {X 0,Y 355.416,Z 985.068,A -85,B 0,C 180,E1 23727.998,E2 23727.998} C_VEL
LIN {X 0,Y 367.057,Z 954.617,A -85,B 0,C 180,E1 23730.321,E2 23730.321} C_VEL
LIN {X 0,Y 362.446,Z 930.938,A -85,B 0,C 180,E1 23735.302,E2 23735.302} C_VEL
LIN {X 0,Y 357.148,Z 912.32,A -85,B 0,C 180,E1 23740.172,E2 23740.172} C_VEL
LIN {X 0,Y 351.302,Z 896.901,A -85,B 0,C 180,E1 23745.652,E2 23745.652} C_VEL
LIN {X 0,Y 346.996,Z 887.115,A -85,B 0,C 180,E1 23750.665,E2 23750.665} C_VEL
LIN {X 0,Y 345.156,Z 882.222,A -85,B 0,C 180,E1 23754.026,E2 23754.026} C_VEL
LIN {X 0,Y 343.752,Z 876.633,A -85,B 0,C 180,E1 23760.009,E2 23760.009} C_VEL
LIN {X 0,Y 343.7,Z 877.671,A -85,B 0,C 180,E1 23763.959,E2 23763.959} C_VEL
LIN {X 0,Y 346.062,Z 884.45,A -85,B 0,C 180,E1 23770.723,E2 23770.723} C_VEL
LIN {X 0,Y 350.539,Z 894.416,A -85,B 0,C 180,E1 23776.416,E2 23776.416} C_VEL
LIN {X 0,Y 350.878,Z 895.324,A -85,B 0,C 180,E1 23776.785,E2 23776.785} C_VEL
LIN {X 0,Y 351.788,Z 902.246,A -85,B 0,C 180,E1 23778.6,E2 23778.6} C_VEL
LIN {X 0,Y 352.653,Z 915.617,A -85,B 0,C 180,E1 23781.47,E2 23781.47} C_VEL
LIN {X 0,Y 358.365,Z 935.624,A -85,B 0,C 180,E1 23787.109,E2 23787.109} C_VEL
LIN {X 0,Y 362.18,Z 957.488,A -85,B 0,C 180,E1 23791.912,E2 23791.912} C_VEL
LIN {X 0,Y 345.252,Z 996.471,A -85,B 0,C 180,E1 23795.025,E2 23795.025} C_VEL
LIN {X 0,Y 326.86,Z 1031.023,A -85,B 0,C 180,E1 23799.067,E2 23799.067} C_VEL
LIN {X 0,Y 307.386,Z 1062.143,A -85,B 0,C 180,E1 23804.382,E2 23804.382} C_VEL
LIN {X 0,Y 289.133,Z 1088.358,A -85,B 0,C 180,E1 23811.039,E2 23811.039} C_VEL
LIN {X 0,Y 273.543,Z 1109.81,A -85,B 0,C 180,E1 23819.295,E2 23819.295} C_VEL
LIN {X 0,Y 262.944,Z 1125.455,A -85,B 0,C 180,E1 23828.894,E2 23828.894} C_VEL
LIN {X 0,Y 258.085,Z 1134.116,A -85,B 0,C 180,E1 23838.146,E2 23838.146} C_VEL
LIN {X 0,Y 256.786,Z 1137.726,A -85,B 0,C 180,E1 23846.62,E2 23846.62} C_VEL
LIN {X 0,Y 256.811,Z 1137.71,A -85,B 0,C 180,E1 23853.385,E2 23853.385} C_VEL
LIN {X 0,Y 258.106,Z 1134.02,A -85,B 0,C 180,E1 23861.859,E2 23861.859} C_VEL
LIN {X 0,Y 263.017,Z 1125.276,A -85,B 0,C 180,E1 23871.106,E2 23871.106} C_VEL
LIN {X 0,Y 272.698,Z 1110.956,A -85,B 0,C 180,E1 23880.007,E2 23880.007} C_VEL
LIN {X 0,Y 288.169,Z 1089.605,A -85,B 0,C 180,E1 23888.445,E2 23888.445} C_VEL
LIN {X 0,Y 306.556,Z 1063.167,A -85,B 0,C 180,E1 23895.278,E2 23895.278} C_VEL
LIN {X 0,Y 325.89,Z 1032.349,A -85,B 0,C 180,E1 23900.623,E2 23900.623} C_VEL
LIN {X 0,Y 344.434,Z 997.767,A -85,B 0,C 180,E1 23904.728,E2 23904.728} C_VEL
LIN {X 0,Y 360.785,Z 960.786,A -85,B 0,C 180,E1 23907.731,E2 23907.731} C_VEL
LIN {X 0,Y 361.989,Z 956.723,A -85,B 0,C 180,E1 23908.112,E2 23908.112} C_VEL
LIN {X 0,Y 357.72,Z 933.676,A -85,B 0,C 180,E1 23913.245,E2 23913.245} C_VEL
LIN {X 0,Y 352.357,Z 915.008,A -85,B 0,C 180,E1 23918.553,E2 23918.553} C_VEL
LIN {X 0,Y 347.166,Z 900.539,A -85,B 0,C 180,E1 23924.136,E2 23924.136} C_VEL
LIN {X 0,Y 342.945,Z 890.052,A -85,B 0,C 180,E1 23930.455,E2 23930.455} C_VEL
LIN {X 0,Y 341.418,Z 884.236,A -85,B 0,C 180,E1 23936.811,E2 23936.811} C_VEL
LIN {X 0,Y 341.488,Z 885.09,A -85,B 0,C 180,E1 23941.42,E2 23941.42} C_VEL
LIN {X 0,Y 343.589,Z 892.118,A -85,B 0,C 180,E1 23947.831,E2 23947.831} C_VEL
LIN {X 0,Y 347.399,Z 901.81,A -85,B 0,C 180,E1 23953.226,E2 23953.226} C_VEL
LIN {X 0,Y 353.006,Z 918.022,A -85,B 0,C 180,E1 23959.211,E2 23959.211} C_VEL
LIN {X 0,Y 358.07,Z 937.117,A -85,B 0,C 180,E1 23964.354,E2 23964.354} C_VEL
LIN {X 0,Y 361.586,Z 958.443,A -85,B 0,C 180,E1 23968.926,E2 23968.926} C_VEL
LIN {X 0,Y 344.896,Z 998.093,A -85,B 0,C 180,E1 23972.097,E2 23972.097} C_VEL
LIN {X 0,Y 325.11,Z 1036.084,A -85,B 0,C 180,E1 23976.489,E2 23976.489} C_VEL
LIN {X 0,Y 304.676,Z 1069.921,A -85,B 0,C 180,E1 23982.287,E2 23982.287} C_VEL
LIN {X 0,Y 286.063,Z 1098.301,A -85,B 0,C 180,E1 23989.543,E2 23989.543} C_VEL
LIN {X 0,Y 271.424,Z 1120.348,A -85,B 0,C 180,E1 23997.97,E2 23997.97} C_VEL
LIN {X 0,Y 261.953,Z 1136.212,A -85,B 0,C 180,E1 24007.204,E2 24007.204} C_VEL
LIN {X 0,Y 257.669,Z 1146.048,A -85,B 0,C 180,E1 24016.393,E2 24016.393} C_VEL
LIN {X 0,Y 256.656,Z 1150.114,A -85,B 0,C 180,E1 24023.216,E2 24023.216} C_VEL
LIN {X 0,Y 256.812,Z 1151.507,A -85,B 0,C 180,E1 24029.997,E2 24029.997} C_VEL
LIN {X 0,Y 256.643,Z 1150.128,A -85,B 0,C 180,E1 24036.778,E2 24036.778} C_VEL
LIN {X 0,Y 258.396,Z 1144.083,A -85,B 0,C 180,E1 24045.92,E2 24045.92} C_VEL
LIN {X 0,Y 264.106,Z 1132.4,A -85,B 0,C 180,E1 24055.482,E2 24055.482} C_VEL
LIN {X 0,Y 275.071,Z 1114.791,A -85,B 0,C 180,E1 24064.532,E2 24064.532} C_VEL
LIN {X 0,Y 290.825,Z 1091.082,A -85,B 0,C 180,E1 24072.628,E2 24072.628} C_VEL
LIN {X 0,Y 308.704,Z 1063.626,A -85,B 0,C 180,E1 24078.989,E2 24078.989} C_VEL
LIN {X 0,Y 327.436,Z 1032.097,A -85,B 0,C 180,E1 24084.071,E2 24084.071} C_VEL
LIN {X 0,Y 345.944,Z 996.122,A -85,B 0,C 180,E1 24088.112,E2 24088.112} C_VEL
LIN {X 0,Y 361.723,Z 957.805,A -85,B 0,C 180,E1 24091.218,E2 24091.218} C_VEL
LIN {X 0,Y 357.907,Z 936.039,A -85,B 0,C 180,E1 24095.967,E2 24095.967} C_VEL
LIN {X 0,Y 352.799,Z 916.831,A -85,B 0,C 180,E1 24101.22,E2 24101.22} C_VEL
LIN {X 0,Y 347.607,Z 902.062,A -85,B 0,C 180,E1 24106.782,E2 24106.782} C_VEL
LIN {X 0,Y 344.205,Z 893.592,A -85,B 0,C 180,E1 24111.467,E2 24111.467} C_VEL
LIN {X 0,Y 342.616,Z 889.422,A -85,B 0,C 180,E1 24114.618,E2 24114.618} C_VEL
LIN {X 0,Y 341.751,Z 884.269,A -85,B 0,C 180,E1 24120.01,E2 24120.01} C_VEL
LIN {X 0,Y 341.634,Z 885.258,A -85,B 0,C 180,E1 24123.824,E2 24123.824} C_VEL
LIN {X 0,Y 343.715,Z 892.054,A -85,B 0,C 180,E1 24130.586,E2 24130.586} C_VEL
LIN {X 0,Y 347.878,Z 902.231,A -85,B 0,C 180,E1 24136.4,E2 24136.4} C_VEL
LIN {X 0,Y 352.653,Z 915.617,A -85,B 0,C 180,E1 24141.47,E2 24141.47} C_VEL
LIN {X 0,Y 353.379,Z 923.507,A -85,B 0,C 180,E1 24143.17,E2 24143.17} C_VEL
LIN {X 0,Y 353.321,Z 938.396,A -85,B 0,C 180,E1 24145.832,E2 24145.832} C_VEL
LIN {X 0,Y 356.793,Z 960.012,A -85,B 0,C 180,E1 24150.864,E2 24150.864} C_VEL
LIN {X 0,Y 352.951,Z 970.569,A -85,B 0,C 180,E1 24151.736,E2 24151.736} C_VEL
LIN {X 0,Y 335.104,Z 1007.826,A -85,B 0,C 180,E1 24155.058,E2 24155.058} C_VEL
LIN {X 0,Y 314.929,Z 1042.589,A -85,B 0,C 180,E1 24159.67,E2 24159.67} C_VEL
LIN {X 0,Y 295.075,Z 1072.068,A -85,B 0,C 180,E1 24165.47,E2 24165.47} C_VEL
LIN {X 0,Y 276.435,Z 1097.161,A -85,B 0,C 180,E1 24172.924,E2 24172.924} C_VEL
LIN {X 0,Y 262.283,Z 1115.897,A -85,B 0,C 180,E1 24181.54,E2 24181.54} C_VEL
LIN {X 0,Y 253.566,Z 1128.511,A -85,B 0,C 180,E1 24190.816,E2 24190.816} C_VEL
LIN {X 0,Y 249.802,Z 1135.4,A -85,B 0,C 180,E1 24199.519,E2 24199.519} C_VEL
LIN {X 0,Y 248.881,Z 1137.933,A -85,B 0,C 180,E1 24206.513,E2 24206.513} C_VEL
LIN {X 0,Y 248.908,Z 1137.917,A -85,B 0,C 180,E1 24213.493,E2 24213.493} C_VEL
LIN {X 0,Y 250.303,Z 1134.23,A -85,B 0,C 180,E1 24222.235,E2 24222.235} C_VEL
LIN {X 0,Y 255.536,Z 1125.492,A -85,B 0,C 180,E1 24231.755,E2 24231.755} C_VEL
LIN {X 0,Y 266.827,Z 1109.748,A -85,B 0,C 180,E1 24241.581,E2 24241.581} C_VEL
LIN {X 0,Y 283.058,Z 1088.229,A -85,B 0,C 180,E1 24249.97,E2 24249.97} C_VEL
LIN {X 0,Y 301.98,Z 1061.916,A -85,B 0,C 180,E1 24256.683,E2 24256.683} C_VEL
LIN {X 0,Y 322.638,Z 1029.685,A -85,B 0,C 180,E1 24262.146,E2 24262.146} C_VEL
LIN {X 0,Y 341.998,Z 993.951,A -85,B 0,C 180,E1 24266.231,E2 24266.231} C_VEL
LIN {X 0,Y 356.671,Z 960.088,A -85,B 0,C 180,E1 24268.99,E2 24268.99} C_VEL
LIN {X 0,Y 353.182,Z 938.581,A -85,B 0,C 180,E1 24273.995,E2 24273.995} C_VEL
LIN {X 0,Y 348.139,Z 919.702,A -85,B 0,C 180,E1 24279.616,E2 24279.616} C_VEL
LIN {X 0,Y 344.029,Z 907.249,A -85,B 0,C 180,E1 24284.669,E2 24284.669} C_VEL
LIN {X 0,Y 340.89,Z 898.794,A -85,B 0,C 180,E1 24289.75,E2 24289.75} C_VEL
LIN {X 0,Y 339.163,Z 891.764,A -85,B 0,C 180,E1 24297.43,E2 24297.43} C_VEL
LIN {X 0,Y 339.261,Z 892.629,A -85,B 0,C 180,E1 24301.246,E2 24301.246} C_VEL
LIN {X 0,Y 341.073,Z 899.541,A -85,B 0,C 180,E1 24307.648,E2 24307.648} C_VEL
LIN {X 0,Y 344.74,Z 909.877,A -85,B 0,C 180,E1 24313.33,E2 24313.33} C_VEL
LIN {X 0,Y 349.922,Z 926.396,A -85,B 0,C 180,E1 24319.387,E2 24319.387} C_VEL
LIN {X 0,Y 354.312,Z 946.956,A -85,B 0,C 180,E1 24324.818,E2 24324.818} C_VEL
LIN {X 0,Y 356.295,Z 961.726,A -85,B 0,C 180,E1 24328.049,E2 24328.049} C_VEL
LIN {X 0,Y 339.531,Z 1000.035,A -85,B 0,C 180,E1 24331.17,E2 24331.17} C_VEL
LIN {X 0,Y 320.21,Z 1036.048,A -85,B 0,C 180,E1 24335.357,E2 24335.357} C_VEL
LIN {X 0,Y 299.123,Z 1069.839,A -85,B 0,C 180,E1 24341.166,E2 24341.166} C_VEL
LIN {X 0,Y 279.869,Z 1098.066,A -85,B 0,C 180,E1 24348.453,E2 24348.453} C_VEL
LIN {X 0,Y 264.531,Z 1120.122,A -85,B 0,C 180,E1 24357.031,E2 24357.031} C_VEL
LIN {X 0,Y 254.561,Z 1135.82,A -85,B 0,C 180,E1 24366.367,E2 24366.367} C_VEL
LIN {X 0,Y 249.863,Z 1145.836,A -85,B 0,C 180,E1 24375.959,E2 24375.959} C_VEL
LIN {X 0,Y 248.754,Z 1149.905,A -85,B 0,C 180,E1 24383,E2 24383} C_VEL
LIN {X 0,Y 248.908,Z 1151.3,A -85,B 0,C 180,E1 24389.997,E2 24389.997} C_VEL
LIN {X 0,Y 248.739,Z 1149.919,A -85,B 0,C 180,E1 24396.995,E2 24396.995} C_VEL
LIN {X 0,Y 250.387,Z 1144.615,A -85,B 0,C 180,E1 24405.618,E2 24405.618} C_VEL
LIN {X 0,Y 256.011,Z 1133.439,A -85,B 0,C 180,E1 24415.406,E2 24415.406} C_VEL
LIN {X 0,Y 267.673,Z 1115.547,A -85,B 0,C 180,E1 24425.084,E2 24425.084} C_VEL
LIN {X 0,Y 283.082,Z 1093.304,A -85,B 0,C 180,E1 24433.03,E2 24433.03} C_VEL
LIN {X 0,Y 301.316,Z 1066.631,A -85,B 0,C 180,E1 24439.509,E2 24439.509} C_VEL
LIN {X 0,Y 321.433,Z 1034.172,A -85,B 0,C 180,E1 24444.92,E2 24444.92} C_VEL
LIN {X 0,Y 340.864,Z 997.707,A -85,B 0,C 180,E1 24449.087,E2 24449.087} C_VEL
LIN {X 0,Y 356.338,Z 962.268,A -85,B 0,C 180,E1 24451.916,E2 24451.916} C_VEL
LIN {X 0,Y 353.624,Z 942.05,A -85,B 0,C 180,E1 24456.414,E2 24456.414} C_VEL
LIN {X 0,Y 349.287,Z 923.739,A -85,B 0,C 180,E1 24461.507,E2 24461.507} C_VEL
LIN {X 0,Y 344.966,Z 910.076,A -85,B 0,C 180,E1 24466.679,E2 24466.679} C_VEL
LIN {X 0,Y 341.264,Z 899.934,A -85,B 0,C 180,E1 24472.356,E2 24472.356} C_VEL
LIN {X 0,Y 340.237,Z 896.824,A -85,B 0,C 180,E1 24474.9,E2 24474.9} C_VEL
LIN {X 0,Y 339.563,Z 891.862,A -85,B 0,C 180,E1 24480.01,E2 24480.01} C_VEL
LIN {X 0,Y 339.407,Z 892.94,A -85,B 0,C 180,E1 24483.769,E2 24483.769} C_VEL
LIN {X 0,Y 341.502,Z 900.56,A -85,B 0,C 180,E1 24491.08,E2 24491.08} C_VEL
LIN {X 0,Y 345.982,Z 912.24,A -85,B 0,C 180,E1 24497.392,E2 24497.392} C_VEL
LIN {X 0,Y 351.184,Z 929.819,A -85,B 0,C 180,E1 24503.451,E2 24503.451} C_VEL
LIN {X 0,Y 353.321,Z 938.396,A -85,B 0,C 180,E1 24505.832,E2 24505.832} C_VEL
LIN {X 0,Y 353.281,Z 947.132,A -85,B 0,C 180,E1 24507.42,E2 24507.42} C_VEL
LIN {X 0,Y 351.558,Z 963.13,A -85,B 0,C 180,E1 24509.907,E2 24509.907} C_VEL
LIN {X 0,Y 350.211,Z 967.857,A -85,B 0,C 180,E1 24510.4,E2 24510.4} C_VEL
LIN {X 0,Y 331.514,Z 1006.417,A -85,B 0,C 180,E1 24513.743,E2 24513.743} C_VEL
LIN {X 0,Y 310.884,Z 1041.28,A -85,B 0,C 180,E1 24518.276,E2 24518.276} C_VEL
LIN {X 0,Y 290.137,Z 1071.262,A -85,B 0,C 180,E1 24524.11,E2 24524.11} C_VEL
LIN {X 0,Y 270.62,Z 1096.647,A -85,B 0,C 180,E1 24531.626,E2 24531.626} C_VEL
LIN {X 0,Y 255.239,Z 1116.114,A -85,B 0,C 180,E1 24540.68,E2 24540.68} C_VEL
LIN {X 0,Y 246.001,Z 1128.723,A -85,B 0,C 180,E1 24550.202,E2 24550.202} C_VEL
LIN {X 0,Y 241.997,Z 1135.608,A -85,B 0,C 180,E1 24559.177,E2 24559.177} C_VEL
LIN {X 0,Y 240.998,Z 1138.14,A -85,B 0,C 180,E1 24566.399,E2 24566.399} C_VEL
LIN {X 0,Y 241.023,Z 1138.125,A -85,B 0,C 180,E1 24573.607,E2 24573.607} C_VEL
LIN {X 0,Y 242.535,Z 1134.439,A -85,B 0,C 180,E1 24582.633,E2 24582.633} C_VEL
LIN {X 0,Y 247.369,Z 1126.708,A -85,B 0,C 180,E1 24591.565,E2 24591.565} C_VEL
LIN {X 0,Y 257.67,Z 1112.887,A -85,B 0,C 180,E1 24600.969,E2 24600.969} C_VEL
LIN {X 0,Y 272.878,Z 1093.617,A -85,B 0,C 180,E1 24609.302,E2 24609.302} C_VEL
LIN {X 0,Y 291.331,Z 1069.395,A -85,B 0,C 180,E1 24616.192,E2 24616.192} C_VEL
LIN {X 0,Y 311.161,Z 1040.584,A -85,B 0,C 180,E1 24621.708,E2 24621.708} C_VEL
LIN {X 0,Y 331.361,Z 1006.476,A -85,B 0,C 180,E1 24626.118,E2 24626.118} C_VEL
LIN {X 0,Y 349.564,Z 968.954,A -85,B 0,C 180,E1 24629.398,E2 24629.398} C_VEL
LIN {X 0,Y 351.392,Z 963.212,A -85,B 0,C 180,E1 24629.955,E2 24629.955} C_VEL
LIN {X 0,Y 348.48,Z 942.834,A -85,B 0,C 180,E1 24634.91,E2 24634.91} C_VEL
LIN {X 0,Y 344.054,Z 924.366,A -85,B 0,C 180,E1 24640.706,E2 24640.706} C_VEL
LIN {X 0,Y 340.065,Z 911.517,A -85,B 0,C 180,E1 24646.477,E2 24646.477} C_VEL
LIN {X 0,Y 337.257,Z 903.779,A -85,B 0,C 180,E1 24652.245,E2 24652.245} C_VEL
LIN {X 0,Y 336.841,Z 899.3,A -85,B 0,C 180,E1 24657.412,E2 24657.412} C_VEL
LIN {X 0,Y 336.921,Z 899.248,A -85,B 0,C 180,E1 24659.99,E2 24659.99} C_VEL
LIN {X 0,Y 338.483,Z 907.265,A -85,B 0,C 180,E1 24667.707,E2 24667.707} C_VEL
LIN {X 0,Y 341.834,Z 917.76,A -85,B 0,C 180,E1 24673.445,E2 24673.445} C_VEL
LIN {X 0,Y 346.369,Z 934.356,A -85,B 0,C 180,E1 24679.473,E2 24679.473} C_VEL
LIN {X 0,Y 350.095,Z 955.248,A -85,B 0,C 180,E1 24684.946,E2 24684.946} C_VEL
LIN {X 0,Y 350.836,Z 965.767,A -85,B 0,C 180,E1 24687.212,E2 24687.212} C_VEL
LIN {X 0,Y 333.59,Z 1003.258,A -85,B 0,C 180,E1 24690.343,E2 24690.343} C_VEL
LIN {X 0,Y 314.316,Z 1037.801,A -85,B 0,C 180,E1 24694.45,E2 24694.45} C_VEL
LIN {X 0,Y 293.15,Z 1070.54,A -85,B 0,C 180,E1 24700.179,E2 24700.179} C_VEL
LIN {X 0,Y 273.758,Z 1097.83,A -85,B 0,C 180,E1 24707.309,E2 24707.309} C_VEL
LIN {X 0,Y 257.468,Z 1120.254,A -85,B 0,C 180,E1 24716.21,E2 24716.21} C_VEL
LIN {X 0,Y 246.625,Z 1136.486,A -85,B 0,C 180,E1 24726.276,E2 24726.276} C_VEL
LIN {X 0,Y 242.113,Z 1145.625,A -85,B 0,C 180,E1 24735.5,E2 24735.5} C_VEL
LIN {X 0,Y 240.874,Z 1149.697,A -85,B 0,C 180,E1 24742.77,E2 24742.77} C_VEL
LIN {X 0,Y 241.014,Z 1151.093,A -85,B 0,C 180,E1 24749.997,E2 24749.997} C_VEL
LIN {X 0,Y 240.859,Z 1149.711,A -85,B 0,C 180,E1 24757.225,E2 24757.225} C_VEL
LIN {X 0,Y 242.698,Z 1144.24,A -85,B 0,C 180,E1 24766.313,E2 24766.313} C_VEL
LIN {X 0,Y 248.685,Z 1133.224,A -85,B 0,C 180,E1 24776.21,E2 24776.21} C_VEL
LIN {X 0,Y 260.196,Z 1116.432,A -85,B 0,C 180,E1 24785.61,E2 24785.61} C_VEL
LIN {X 0,Y 276.267,Z 1094.297,A -85,B 0,C 180,E1 24793.817,E2 24793.817} C_VEL
LIN {X 0,Y 295.009,Z 1068.008,A -85,B 0,C 180,E1 24800.385,E2 24800.385} C_VEL
LIN {X 0,Y 315.413,Z 1036.307,A -85,B 0,C 180,E1 24805.798,E2 24805.798} C_VEL
LIN {X 0,Y 336.535,Z 997.874,A -85,B 0,C 180,E1 24810.222,E2 24810.222} C_VEL
LIN {X 0,Y 351.224,Z 965.294,A -85,B 0,C 180,E1 24812.842,E2 24812.842} C_VEL
LIN {X 0,Y 348.575,Z 944.582,A -85,B 0,C 180,E1 24817.73,E2 24817.73} C_VEL
LIN {X 0,Y 344.88,Z 927.657,A -85,B 0,C 180,E1 24822.792,E2 24822.792} C_VEL
LIN {X 0,Y 340.905,Z 914.205,A -85,B 0,C 180,E1 24828.344,E2 24828.344} C_VEL
LIN {X 0,Y 337.705,Z 904.343,A -85,B 0,C 180,E1 24834.862,E2 24834.862} C_VEL
LIN {X 0,Y 337.223,Z 899.425,A -85,B 0,C 180,E1 24840.01,E2 24840.01} C_VEL
LIN {X 0,Y 337.018,Z 900.35,A -85,B 0,C 180,E1 24843.553,E2 24843.553} C_VEL
LIN {X 0,Y 338.941,Z 908.296,A -85,B 0,C 180,E1 24851.165,E2 24851.165} C_VEL
LIN {X 0,Y 342.863,Z 919.835,A -85,B 0,C 180,E1 24857.363,E2 24857.363} C_VEL
LIN {X 0,Y 347.522,Z 937.646,A -85,B 0,C 180,E1 24863.477,E2 24863.477} C_VEL
LIN {X 0,Y 350.868,Z 956.362,A -85,B 0,C 180,E1 24868.368,E2 24868.368} C_VEL
LIN {X 0,Y 351.558,Z 963.13,A -85,B 0,C 180,E1 24869.907,E2 24869.907} C_VEL
LIN {X 0,Y 349.752,Z 968.277,A -85,B 0,C 180,E1 24870.346,E2 24870.346} C_VEL
LIN {X 0,Y 339.728,Z 982.561,A -85,B 0,C 180,E1 24870.373,E2 24870.373} C_VEL
LIN {X 0,Y 339.382,Z 983.221,A -85,B 0,C 180,E1 24870.425,E2 24870.425} C_VEL
LIN {X 0,Y 319.92,Z 1019.416,A -85,B 0,C 180,E1 24874.027,E2 24874.027} C_VEL
LIN {X 0,Y 297.823,Z 1053.416,A -85,B 0,C 180,E1 24879.123,E2 24879.123} C_VEL
LIN {X 0,Y 276.237,Z 1082.237,A -85,B 0,C 180,E1 24885.761,E2 24885.761} C_VEL
LIN {X 0,Y 257.44,Z 1105.161,A -85,B 0,C 180,E1 24893.949,E2 24893.949} C_VEL
LIN {X 0,Y 244.045,Z 1121.595,A -85,B 0,C 180,E1 24903.252,E2 24903.252} C_VEL
LIN {X 0,Y 236.141,Z 1132.333,A -85,B 0,C 180,E1 24913.413,E2 24913.413} C_VEL
LIN {X 0,Y 233.36,Z 1137.404,A -85,B 0,C 180,E1 24922.542,E2 24922.542} C_VEL
LIN {X 0,Y 233.216,Z 1138.655,A -85,B 0,C 180,E1 24930.003,E2 24930.003} C_VEL
LIN {X 0,Y 233.404,Z 1137.364,A -85,B 0,C 180,E1 24937.463,E2 24937.463} C_VEL
LIN {X 0,Y 236.29,Z 1132.064,A -85,B 0,C 180,E1 24946.773,E2 24946.773} C_VEL
LIN {X 0,Y 244.11,Z 1121.393,A -85,B 0,C 180,E1 24956.747,E2 24956.747} C_VEL
LIN {X 0,Y 257.59,Z 1104.907,A -85,B 0,C 180,E1 24966.033,E2 24966.033} C_VEL
LIN {X 0,Y 276.517,Z 1081.698,A -85,B 0,C 180,E1 24974.279,E2 24974.279} C_VEL
LIN {X 0,Y 298.015,Z 1052.95,A -85,B 0,C 180,E1 24980.84,E2 24980.84} C_VEL
LIN {X 0,Y 319.498,Z 1019.857,A -85,B 0,C 180,E1 24985.79,E2 24985.79} C_VEL
LIN {X 0,Y 339.464,Z 982.496,A -85,B 0,C 180,E1 24989.545,E2 24989.545} C_VEL
LIN {X 0,Y 345.909,Z 968.643,A -85,B 0,C 180,E1 24990.578,E2 24990.578} C_VEL
LIN {X 0,Y 345.12,Z 955.3,A -85,B 0,C 180,E1 24993.627,E2 24993.627} C_VEL
LIN {X 0,Y 341.618,Z 936.224,A -85,B 0,C 180,E1 24999.209,E2 24999.209} C_VEL
LIN {X 0,Y 337.905,Z 921.724,A -85,B 0,C 180,E1 25005.05,E2 25005.05} C_VEL
LIN {X 0,Y 335.272,Z 913.101,A -85,B 0,C 180,E1 25010.498,E2 25010.498} C_VEL
LIN {X 0,Y 334.311,Z 906.793,A -85,B 0,C 180,E1 25017.393,E2 25017.393} C_VEL
LIN {X 0,Y 334.365,Z 906.811,A -85,B 0,C 180,E1 25019.99,E2 25019.99} C_VEL
LIN {X 0,Y 335.479,Z 913.739,A -85,B 0,C 180,E1 25026.977,E2 25026.977} C_VEL
LIN {X 0,Y 338.408,Z 924.252,A -85,B 0,C 180,E1 25032.925,E2 25032.925} C_VEL
LIN {X 0,Y 342.291,Z 940.12,A -85,B 0,C 180,E1 25038.879,E2 25038.879} C_VEL
LIN {X 0,Y 345.305,Z 960.856,A -85,B 0,C 180,E1 25044.485,E2 25044.485} C_VEL
LIN {X 0,Y 345.455,Z 969.632,A -85,B 0,C 180,E1 25046.315,E2 25046.315} C_VEL
LIN {X 0,Y 325.528,Z 1010.614,A -85,B 0,C 180,E1 25049.896,E2 25049.896} C_VEL
LIN {X 0,Y 304.457,Z 1045.999,A -85,B 0,C 180,E1 25054.487,E2 25054.487} C_VEL
LIN {X 0,Y 283.882,Z 1075.882,A -85,B 0,C 180,E1 25060.194,E2 25060.194} C_VEL
LIN {X 0,Y 264.947,Z 1101.298,A -85,B 0,C 180,E1 25067.403,E2 25067.403} C_VEL
LIN {X 0,Y 249.505,Z 1121.608,A -85,B 0,C 180,E1 25076.001,E2 25076.001} C_VEL
LIN {X 0,Y 239.071,Z 1136.495,A -85,B 0,C 180,E1 25085.669,E2 25085.669} C_VEL
LIN {X 0,Y 234.019,Z 1146.167,A -85,B 0,C 180,E1 25096.131,E2 25096.131} C_VEL
LIN {X 0,Y 232.849,Z 1150.522,A -85,B 0,C 180,E1 25106.266,E2 25106.266} C_VEL
LIN {X 0,Y 233.108,Z 1150.885,A -85,B 0,C 180,E1 25109.997,E2 25109.997} C_VEL
LIN {X 0,Y 232.96,Z 1149.503,A -85,B 0,C 180,E1 25117.471,E2 25117.471} C_VEL
LIN {X 0,Y 234.987,Z 1144.028,A -85,B 0,C 180,E1 25126.864,E2 25126.864} C_VEL
LIN {X 0,Y 242.239,Z 1131.805,A -85,B 0,C 180,E1 25137.929,E2 25137.929} C_VEL
LIN {X 0,Y 254.982,Z 1114.426,A -85,B 0,C 180,E1 25147.519,E2 25147.519} C_VEL
LIN {X 0,Y 273.25,Z 1090.384,A -85,B 0,C 180,E1 25156.12,E2 25156.12} C_VEL
LIN {X 0,Y 293.264,Z 1062.876,A -85,B 0,C 180,E1 25162.59,E2 25162.59} C_VEL
LIN {X 0,Y 313.406,Z 1031.849,A -85,B 0,C 180,E1 25167.596,E2 25167.596} C_VEL
LIN {X 0,Y 333.179,Z 996.357,A -85,B 0,C 180,E1 25171.535,E2 25171.535} C_VEL
LIN {X 0,Y 346.095,Z 968.084,A -85,B 0,C 180,E1 25173.876,E2 25173.876} C_VEL
LIN {X 0,Y 343.49,Z 946.322,A -85,B 0,C 180,E1 25179.348,E2 25179.348} C_VEL
LIN {X 0,Y 339.863,Z 928.845,A -85,B 0,C 180,E1 25185.158,E2 25185.158} C_VEL
LIN {X 0,Y 336.52,Z 917.118,A -85,B 0,C 180,E1 25190.944,E2 25190.944} C_VEL
LIN {X 0,Y 334.705,Z 910.891,A -85,B 0,C 180,E1 25196.117,E2 25196.117} C_VEL
LIN {X 0,Y 334.649,Z 907.042,A -85,B 0,C 180,E1 25200.01,E2 25200.01} C_VEL
LIN {X 0,Y 334.615,Z 907.003,A -85,B 0,C 180,E1 25202.605,E2 25202.605} C_VEL
LIN {X 0,Y 335.837,Z 914.713,A -85,B 0,C 180,E1 25210.406,E2 25210.406} C_VEL
LIN {X 0,Y 339.402,Z 926.357,A -85,B 0,C 180,E1 25216.877,E2 25216.877} C_VEL
LIN {X 0,Y 343.299,Z 943.612,A -85,B 0,C 180,E1 25222.98,E2 25222.98} C_VEL
LIN {X 0,Y 345.933,Z 961.342,A -85,B 0,C 180,E1 25227.76,E2 25227.76} C_VEL
LIN {X 0,Y 346.38,Z 967.976,A -85,B 0,C 180,E1 25229.252,E2 25229.252} C_VEL
LIN {X 0,Y 339.382,Z 983.221,A -85,B 0,C 180,E1 25230.425,E2 25230.425} C_VEL
LIN {X 0,Y 330.049,Z 997.638,A -85,B 0,C 180,E1 25231.085,E2 25231.085} C_VEL
LIN {X 0,Y 321.377,Z 1009.77,A -85,B 0,C 180,E1 25231.704,E2 25231.704} C_VEL
LIN {X 0,Y 320.367,Z 1011.409,A -85,B 0,C 180,E1 25231.878,E2 25231.878} C_VEL
LIN {X 0,Y 300.163,Z 1043.346,A -85,B 0,C 180,E1 25236.138,E2 25236.138} C_VEL
LIN {X 0,Y 278.136,Z 1073.116,A -85,B 0,C 180,E1 25242.082,E2 25242.082} C_VEL
LIN {X 0,Y 257.556,Z 1097.822,A -85,B 0,C 180,E1 25249.68,E2 25249.68} C_VEL
LIN {X 0,Y 241.131,Z 1116.814,A -85,B 0,C 180,E1 25258.969,E2 25258.969} C_VEL
LIN {X 0,Y 230.988,Z 1129.145,A -85,B 0,C 180,E1 25268.856,E2 25268.856} C_VEL
LIN {X 0,Y 226.396,Z 1136.024,A -85,B 0,C 180,E1 25278.421,E2 25278.421} C_VEL
LIN {X 0,Y 225.214,Z 1138.555,A -85,B 0,C 180,E1 25286.146,E2 25286.146} C_VEL
LIN {X 0,Y 225.238,Z 1138.54,A -85,B 0,C 180,E1 25293.861,E2 25293.861} C_VEL
LIN {X 0,Y 226.985,Z 1134.903,A -85,B 0,C 180,E1 25303.442,E2 25303.442} C_VEL
LIN {X 0,Y 233.456,Z 1125.932,A -85,B 0,C 180,E1 25314.121,E2 25314.121} C_VEL
LIN {X 0,Y 246.738,Z 1110.22,A -85,B 0,C 180,E1 25324.616,E2 25324.616} C_VEL
LIN {X 0,Y 265.02,Z 1088.927,A -85,B 0,C 180,E1 25333.323,E2 25333.323} C_VEL
LIN {X 0,Y 286.139,Z 1062.489,A -85,B 0,C 180,E1 25340.229,E2 25340.229} C_VEL
LIN {X 0,Y 308.493,Z 1030.612,A -85,B 0,C 180,E1 25345.645,E2 25345.645} C_VEL
LIN {X 0,Y 330.034,Z 993.568,A -85,B 0,C 180,E1 25349.806,E2 25349.806} C_VEL
LIN {X 0,Y 340.757,Z 971.821,A -85,B 0,C 180,E1 25351.529,E2 25351.529} C_VEL
LIN {X 0,Y 340.073,Z 957.812,A -85,B 0,C 180,E1 25354.94,E2 25354.94} C_VEL
LIN {X 0,Y 337.045,Z 939.504,A -85,B 0,C 180,E1 25360.748,E2 25360.748} C_VEL
LIN {X 0,Y 334.145,Z 927.102,A -85,B 0,C 180,E1 25366.219,E2 25366.219} C_VEL
LIN {X 0,Y 331.826,Z 918.867,A -85,B 0,C 180,E1 25372.117,E2 25372.117} C_VEL
LIN {X 0,Y 331.63,Z 914.295,A -85,B 0,C 180,E1 25377.372,E2 25377.372} C_VEL
LIN {X 0,Y 331.666,Z 914.348,A -85,B 0,C 180,E1 25379.99,E2 25379.99} C_VEL
LIN {X 0,Y 332.823,Z 922.481,A -85,B 0,C 180,E1 25387.839,E2 25387.839} C_VEL
LIN {X 0,Y 335.52,Z 933.49,A -85,B 0,C 180,E1 25393.703,E2 25393.703} C_VEL
LIN {X 0,Y 338.693,Z 950.067,A -85,B 0,C 180,E1 25399.593,E2 25399.593} C_VEL
LIN {X 0,Y 340.778,Z 970.742,A -85,B 0,C 180,E1 25405.031,E2 25405.031} C_VEL
LIN {X 0,Y 338.511,Z 976.747,A -85,B 0,C 180,E1 25405.654,E2 25405.654} C_VEL
LIN {X 0,Y 319.506,Z 1013.847,A -85,B 0,C 180,E1 25409.028,E2 25409.028} C_VEL
LIN {X 0,Y 298.048,Z 1048.534,A -85,B 0,C 180,E1 25413.648,E2 25413.648} C_VEL
LIN {X 0,Y 276.022,Z 1079.314,A -85,B 0,C 180,E1 25419.777,E2 25419.777} C_VEL
LIN {X 0,Y 255.991,Z 1104.806,A -85,B 0,C 180,E1 25427.501,E2 25427.501} C_VEL
LIN {X 0,Y 240.454,Z 1124.267,A -85,B 0,C 180,E1 25436.536,E2 25436.536} C_VEL
LIN {X 0,Y 230.293,Z 1138.382,A -85,B 0,C 180,E1 25446.746,E2 25446.746} C_VEL
LIN {X 0,Y 226.136,Z 1146.189,A -85,B 0,C 180,E1 25456.004,E2 25456.004} C_VEL
LIN {X 0,Y 224.937,Z 1150.315,A -85,B 0,C 180,E1 25466.134,E2 25466.134} C_VEL
LIN {X 0,Y 225.228,Z 1150.679,A -85,B 0,C 180,E1 25469.997,E2 25469.997} C_VEL
LIN {X 0,Y 225.064,Z 1149.294,A -85,B 0,C 180,E1 25477.735,E2 25477.735} C_VEL
LIN {X 0,Y 227.269,Z 1143.816,A -85,B 0,C 180,E1 25487.455,E2 25487.455} C_VEL
LIN {X 0,Y 234.97,Z 1131.772,A -85,B 0,C 180,E1 25498.732,E2 25498.732} C_VEL
LIN {X 0,Y 248.527,Z 1114.203,A -85,B 0,C 180,E1 25508.671,E2 25508.671} C_VEL
LIN {X 0,Y 267.676,Z 1090.154,A -85,B 0,C 180,E1 25517.375,E2 25517.375} C_VEL
LIN {X 0,Y 288.37,Z 1062.624,A -85,B 0,C 180,E1 25523.881,E2 25523.881} C_VEL
LIN {X 0,Y 309.411,Z 1031.14,A -85,B 0,C 180,E1 25528.918,E2 25528.918} C_VEL
LIN {X 0,Y 329.341,Z 996.189,A -85,B 0,C 180,E1 25532.75,E2 25532.75} C_VEL
LIN {X 0,Y 340.975,Z 971.58,A -85,B 0,C 180,E1 25534.805,E2 25534.805} C_VEL
LIN {X 0,Y 339.037,Z 951.436,A -85,B 0,C 180,E1 25540.066,E2 25540.066} C_VEL
LIN {X 0,Y 336.102,Z 935.173,A -85,B 0,C 180,E1 25545.656,E2 25545.656} C_VEL
LIN {X 0,Y 333.581,Z 924.759,A -85,B 0,C 180,E1 25550.863,E2 25550.863} C_VEL
LIN {X 0,Y 331.848,Z 918.318,A -85,B 0,C 180,E1 25556.083,E2 25556.083} C_VEL
LIN {X 0,Y 331.937,Z 914.583,A -85,B 0,C 180,E1 25560.01,E2 25560.01} C_VEL
LIN {X 0,Y 331.902,Z 914.558,A -85,B 0,C 180,E1 25562.626,E2 25562.626} C_VEL
LIN {X 0,Y 332.933,Z 922.307,A -85,B 0,C 180,E1 25570.497,E2 25570.497} C_VEL
LIN {X 0,Y 335.707,Z 932.748,A -85,B 0,C 180,E1 25576.393,E2 25576.393} C_VEL
LIN {X 0,Y 338.968,Z 949.299,A -85,B 0,C 180,E1 25582.417,E2 25582.417} C_VEL
LIN {X 0,Y 341.114,Z 967.139,A -85,B 0,C 180,E1 25587.337,E2 25587.337} C_VEL
LIN {X 0,Y 340.75,Z 972.259,A -85,B 0,C 180,E1 25588.384,E2 25588.384} C_VEL
LIN {X 0,Y 321.602,Z 1009.3,A -85,B 0,C 180,E1 25591.64,E2 25591.64} C_VEL
LIN {X 0,Y 320.367,Z 1011.409,A -85,B 0,C 180,E1 25591.878,E2 25591.878} C_VEL
LIN {X 0,Y 310.234,Z 1024.771,A -85,B 0,C 180,E1 25592.845,E2 25592.845} C_VEL
LIN {X 0,Y 300.837,Z 1035.949,A -85,B 0,C 180,E1 25593.737,E2 25593.737} C_VEL
LIN {X 0,Y 299.753,Z 1037.459,A -85,B 0,C 180,E1 25593.948,E2 25593.948} C_VEL
LIN {X 0,Y 279.12,Z 1065.402,A -85,B 0,C 180,E1 25598.977,E2 25598.977} C_VEL
LIN {X 0,Y 258.056,Z 1090.616,A -85,B 0,C 180,E1 25605.799,E2 25605.799} C_VEL
LIN {X 0,Y 239.994,Z 1110.694,A -85,B 0,C 180,E1 25614.273,E2 25614.273} C_VEL
LIN {X 0,Y 226.047,Z 1126.375,A -85,B 0,C 180,E1 25625.098,E2 25625.098} C_VEL
LIN {X 0,Y 219.567,Z 1134.618,A -85,B 0,C 180,E1 25635.075,E2 25635.075} C_VEL
LIN {X 0,Y 217.31,Z 1138.762,A -85,B 0,C 180,E1 25646.005,E2 25646.005} C_VEL
LIN {X 0,Y 217.335,Z 1138.747,A -85,B 0,C 180,E1 25654.001,E2 25654.001} C_VEL
LIN {X 0,Y 219.634,Z 1134.491,A -85,B 0,C 180,E1 25664.991,E2 25664.991} C_VEL
LIN {X 0,Y 227.256,Z 1124.825,A -85,B 0,C 180,E1 25676.074,E2 25676.074} C_VEL
LIN {X 0,Y 240.136,Z 1110.443,A -85,B 0,C 180,E1 25685.711,E2 25685.711} C_VEL
LIN {X 0,Y 259.243,Z 1089.158,A -85,B 0,C 180,E1 25694.539,E2 25694.539} C_VEL
LIN {X 0,Y 281.34,Z 1062.401,A -85,B 0,C 180,E1 25701.551,E2 25701.551} C_VEL
LIN {X 0,Y 303.632,Z 1031.538,A -85,B 0,C 180,E1 25706.797,E2 25706.797} C_VEL
LIN {X 0,Y 325.185,Z 995.632,A -85,B 0,C 180,E1 25710.854,E2 25710.854} C_VEL
LIN {X 0,Y 335.74,Z 974.896,A -85,B 0,C 180,E1 25712.521,E2 25712.521} C_VEL
LIN {X 0,Y 334.885,Z 958.501,A -85,B 0,C 180,E1 25716.897,E2 25716.897} C_VEL
LIN {X 0,Y 332.361,Z 941.864,A -85,B 0,C 180,E1 25722.756,E2 25722.756} C_VEL
LIN {X 0,Y 329.922,Z 930.874,A -85,B 0,C 180,E1 25728.431,E2 25728.431} C_VEL
LIN {X 0,Y 328.602,Z 922.688,A -85,B 0,C 180,E1 25736.024,E2 25736.024} C_VEL
LIN {X 0,Y 328.768,Z 921.794,A -85,B 0,C 180,E1 25739.99,E2 25739.99} C_VEL
LIN {X 0,Y 329.397,Z 928.141,A -85,B 0,C 180,E1 25746.593,E2 25746.593} C_VEL
LIN {X 0,Y 331.498,Z 938.375,A -85,B 0,C 180,E1 25752.528,E2 25752.528} C_VEL
LIN {X 0,Y 334.155,Z 954.039,A -85,B 0,C 180,E1 25758.494,E2 25758.494} C_VEL
LIN {X 0,Y 335.646,Z 973.705,A -85,B 0,C 180,E1 25763.958,E2 25763.958} C_VEL
LIN {X 0,Y 334.466,Z 977.714,A -85,B 0,C 180,E1 25764.51,E2 25764.51} C_VEL
LIN {X 0,Y 314.959,Z 1014.711,A -85,B 0,C 180,E1 25767.871,E2 25767.871} C_VEL
LIN {X 0,Y 293.628,Z 1048.265,A -85,B 0,C 180,E1 25772.326,E2 25772.326} C_VEL
LIN {X 0,Y 270.855,Z 1079.069,A -85,B 0,C 180,E1 25778.445,E2 25778.445} C_VEL
LIN {X 0,Y 249.242,Z 1105.552,A -85,B 0,C 180,E1 25786.597,E2 25786.597} C_VEL
LIN {X 0,Y 232.448,Z 1125.621,A -85,B 0,C 180,E1 25796.351,E2 25796.351} C_VEL
LIN {X 0,Y 222.302,Z 1138.967,A -85,B 0,C 180,E1 25806.713,E2 25806.713} C_VEL
LIN {X 0,Y 217.788,Z 1147.367,A -85,B 0,C 180,E1 25817.95,E2 25817.95} C_VEL
LIN {X 0,Y 217.025,Z 1150.107,A -85,B 0,C 180,E1 25825.993,E2 25825.993} C_VEL
LIN {X 0,Y 217.32,Z 1150.471,A -85,B 0,C 180,E1 25829.997,E2 25829.997} C_VEL
LIN {X 0,Y 217.17,Z 1149.085,A -85,B 0,C 180,E1 25838.018,E2 25838.018} C_VEL
LIN {X 0,Y 219.582,Z 1143.603,A -85,B 0,C 180,E1 25848.086,E2 25848.086} C_VEL
LIN {X 0,Y 227.445,Z 1132.097,A -85,B 0,C 180,E1 25859.319,E2 25859.319} C_VEL
LIN {X 0,Y 242.195,Z 1113.983,A -85,B 0,C 180,E1 25869.88,E2 25869.88} C_VEL
LIN {X 0,Y 262.211,Z 1089.922,A -85,B 0,C 180,E1 25878.689,E2 25878.689} C_VEL
LIN {X 0,Y 283.586,Z 1062.445,A -85,B 0,C 180,E1 25885.198,E2 25885.198} C_VEL
LIN {X 0,Y 304.703,Z 1031.808,A -85,B 0,C 180,E1 25890.1,E2 25890.1} C_VEL
LIN {X 0,Y 325.015,Z 997.243,A -85,B 0,C 180,E1 25893.893,E2 25893.893} C_VEL
LIN {X 0,Y 335.688,Z 975.713,A -85,B 0,C 180,E1 25895.643,E2 25895.643} C_VEL
LIN {X 0,Y 334.642,Z 957.008,A -85,B 0,C 180,E1 25900.666,E2 25900.666} C_VEL
LIN {X 0,Y 332.229,Z 940.926,A -85,B 0,C 180,E1 25906.418,E2 25906.418} C_VEL
LIN {X 0,Y 329.887,Z 930.398,A -85,B 0,C 180,E1 25912.091,E2 25912.091} C_VEL
LIN {X 0,Y 328.78,Z 923.418,A -85,B 0,C 180,E1 25918.69,E2 25918.69} C_VEL
LIN {X 0,Y 329.027,Z 922.058,A -85,B 0,C 180,E1 25920.01,E2 25920.01} C_VEL
LIN {X 0,Y 328.987,Z 922.055,A -85,B 0,C 180,E1 25922.649,E2 25922.649} C_VEL
LIN {X 0,Y 329.855,Z 929.852,A -85,B 0,C 180,E1 25930.597,E2 25930.597} C_VEL
LIN {X 0,Y 332.465,Z 941.353,A -85,B 0,C 180,E1 25936.862,E2 25936.862} C_VEL
LIN {X 0,Y 335.049,Z 958.535,A -85,B 0,C 180,E1 25942.965,E2 25942.965} C_VEL
LIN {X 0,Y 336.164,Z 974.114,A -85,B 0,C 180,E1 25947.248,E2 25947.248} C_VEL
LIN {X 0,Y 317.328,Z 1009.867,A -85,B 0,C 180,E1 25950.447,E2 25950.447} C_VEL
LIN {X 0,Y 299.753,Z 1037.459,A -85,B 0,C 180,E1 25953.948,E2 25953.948} C_VEL
LIN {X 0,Y 288.838,Z 1049.628,A -85,B 0,C 180,E1 25955.223,E2 25955.223} C_VEL
LIN {X 0,Y 278.903,Z 1059.692,A -85,B 0,C 180,E1 25956.429,E2 25956.429} C_VEL
LIN {X 0,Y 277.793,Z 1061.064,A -85,B 0,C 180,E1 25956.691,E2 25956.691} C_VEL
LIN {X 0,Y 255.979,Z 1086.811,A -85,B 0,C 180,E1 25963.239,E2 25963.239} C_VEL
LIN {X 0,Y 236.651,Z 1107.512,A -85,B 0,C 180,E1 25971.377,E2 25971.377} C_VEL
LIN {X 0,Y 221.651,Z 1123.386,A -85,B 0,C 180,E1 25981.416,E2 25981.416} C_VEL
LIN {X 0,Y 212.328,Z 1134.206,A -85,B 0,C 180,E1 25993.419,E2 25993.419} C_VEL
LIN {X 0,Y 209.775,Z 1138.027,A -85,B 0,C 180,E1 26001.698,E2 26001.698} C_VEL
LIN {X 0,Y 209.557,Z 1139.276,A -85,B 0,C 180,E1 26010.004,E2 26010.004} C_VEL
LIN {X 0,Y 209.814,Z 1137.988,A -85,B 0,C 180,E1 26018.308,E2 26018.308} C_VEL
LIN {X 0,Y 213.429,Z 1132.696,A -85,B 0,C 180,E1 26028.634,E2 26028.634} C_VEL
LIN {X 0,Y 222.846,Z 1122.043,A -85,B 0,C 180,E1 26039.538,E2 26039.538} C_VEL
LIN {X 0,Y 239.582,Z 1104.431,A -85,B 0,C 180,E1 26049.971,E2 26049.971} C_VEL
LIN {X 0,Y 260.987,Z 1081.039,A -85,B 0,C 180,E1 26058.376,E2 26058.376} C_VEL
LIN {X 0,Y 283.47,Z 1053.697,A -85,B 0,C 180,E1 26064.604,E2 26064.604} C_VEL
LIN {X 0,Y 307.391,Z 1019.648,A -85,B 0,C 180,E1 26069.614,E2 26069.614} C_VEL
LIN {X 0,Y 328.408,Z 982.893,A -85,B 0,C 180,E1 26073.166,E2 26073.166} C_VEL
LIN {X 0,Y 330.816,Z 978.037,A -85,B 0,C 180,E1 26073.529,E2 26073.529} C_VEL
LIN {X 0,Y 330.025,Z 960.958,A -85,B 0,C 180,E1 26078.443,E2 26078.443} C_VEL
LIN {X 0,Y 328.156,Z 946.545,A -85,B 0,C 180,E1 26083.908,E2 26083.908} C_VEL
LIN {X 0,Y 326.346,Z 937,A -85,B 0,C 180,E1 26089.288,E2 26089.288} C_VEL
LIN {X 0,Y 325.728,Z 929.096,A -85,B 0,C 180,E1 26097.324,E2 26097.324} C_VEL
LIN {X 0,Y 325.74,Z 929.184,A -85,B 0,C 180,E1 26099.99,E2 26099.99} C_VEL
LIN {X 0,Y 326.118,Z 935.601,A -85,B 0,C 180,E1 26106.659,E2 26106.659} C_VEL
LIN {X 0,Y 327.923,Z 946.064,A -85,B 0,C 180,E1 26112.667,E2 26112.667} C_VEL
LIN {X 0,Y 329.941,Z 962.25,A -85,B 0,C 180,E1 26118.739,E2 26118.739} C_VEL
LIN {X 0,Y 330.615,Z 977.696,A -85,B 0,C 180,E1 26123.109,E2 26123.109} C_VEL
LIN {X 0,Y 327.239,Z 985.522,A -85,B 0,C 180,E1 26123.867,E2 26123.867} C_VEL
LIN {X 0,Y 305.638,Z 1023.703,A -85,B 0,C 180,E1 26127.602,E2 26127.602} C_VEL
LIN {X 0,Y 281.583,Z 1058.652,A -85,B 0,C 180,E1 26132.779,E2 26132.779} C_VEL
LIN {X 0,Y 258.053,Z 1088.292,A -85,B 0,C 180,E1 26139.585,E2 26139.585} C_VEL
LIN {X 0,Y 237.618,Z 1111.734,A -85,B 0,C 180,E1 26147.965,E2 26147.965} C_VEL
LIN {X 0,Y 223.195,Z 1128.246,A -85,B 0,C 180,E1 26157.102,E2 26157.102} C_VEL
LIN {X 0,Y 213.579,Z 1140.774,A -85,B 0,C 180,E1 26167.961,E2 26167.961} C_VEL
LIN {X 0,Y 209.975,Z 1147.157,A -85,B 0,C 180,E1 26177.494,E2 26177.494} C_VEL
LIN {X 0,Y 209.112,Z 1149.899,A -85,B 0,C 180,E1 26185.841,E2 26185.841} C_VEL
LIN {X 0,Y 209.437,Z 1150.265,A -85,B 0,C 180,E1 26189.996,E2 26189.996} C_VEL
LIN {X 0,Y 209.285,Z 1148.877,A -85,B 0,C 180,E1 26198.322,E2 26198.322} C_VEL
LIN {X 0,Y 211.937,Z 1143.391,A -85,B 0,C 180,E1 26208.763,E2 26208.763} C_VEL
LIN {X 0,Y 220.218,Z 1132.058,A -85,B 0,C 180,E1 26220.212,E2 26220.212} C_VEL
LIN {X 0,Y 235.985,Z 1113.762,A -85,B 0,C 180,E1 26231.152,E2 26231.152} C_VEL
LIN {X 0,Y 256.929,Z 1089.693,A -85,B 0,C 180,E1 26240.048,E2 26240.048} C_VEL
LIN {X 0,Y 279.526,Z 1061.525,A -85,B 0,C 180,E1 26246.705,E2 26246.705} C_VEL
LIN {X 0,Y 301.746,Z 1029.961,A -85,B 0,C 180,E1 26251.643,E2 26251.643} C_VEL
LIN {X 0,Y 322.875,Z 994.396,A -85,B 0,C 180,E1 26255.391,E2 26255.391} C_VEL
LIN {X 0,Y 330.791,Z 978.021,A -85,B 0,C 180,E1 26256.851,E2 26256.851} C_VEL
LIN {X 0,Y 329.888,Z 959.683,A -85,B 0,C 180,E1 26262.159,E2 26262.159} C_VEL
LIN {X 0,Y 327.897,Z 944.866,A -85,B 0,C 180,E1 26268.01,E2 26268.01} C_VEL
LIN {X 0,Y 326.288,Z 935.963,A -85,B 0,C 180,E1 26273.344,E2 26273.344} C_VEL
LIN {X 0,Y 325.976,Z 929.469,A -85,B 0,C 180,E1 26280.01,E2 26280.01} C_VEL
LIN {X 0,Y 325.934,Z 929.477,A -85,B 0,C 180,E1 26282.674,E2 26282.674} C_VEL
LIN {X 0,Y 326.602,Z 937.338,A -85,B 0,C 180,E1 26290.703,E2 26290.703} C_VEL
LIN {X 0,Y 328.563,Z 948.034,A -85,B 0,C 180,E1 26296.569,E2 26296.569} C_VEL
LIN {X 0,Y 330.538,Z 964.745,A -85,B 0,C 180,E1 26302.606,E2 26302.606} C_VEL
LIN {X 0,Y 330.833,Z 978.487,A -85,B 0,C 180,E1 26306.392,E2 26306.392} C_VEL
